IF GVL.g_stTrackingSimulation.Mode <> E_ApplicationSimulationMode.SIM_OFF AND GVL.g_stTrackingSimulation.VirtualEncoderEnable THEN 
	SMC_FreeEncoder.diEncoderPosition := diVirtualEncoderA; 
ELSE
	//SMC_FreeEncoder.diEncoderPosition := TO_DINT(AXIS_6.fActPosition);
	//SMC_FreeEncoder.diEncoderPosition :=AXIS_6.diActPosition;
// 	IF udiv < 400 THEN
// 		SMC_FreeEncoder.diEncoderPosition := SMC_FreeEncoder.diEncoderPosition - 10;
// 	END_IF
// 	IF udiv >= 400 THEN
// 		SMC_FreeEncoder.diEncoderPosition := SMC_FreeEncoder.diEncoderPosition - 11;
// 	END_IF
// 	IF udiv = 3 THEN
// 		SMC_FreeEncoder.diEncoderPosition := SMC_FreeEncoder.diEncoderPosition - 5;
// 	END_IF
// 	IF udiv = 4 THEN
// 		SMC_FreeEncoder.diEncoderPosition := SMC_FreeEncoder.diEncoderPosition - 5;
// 	END_IF
	IF GVL.Y[10] <> FALSE THEN
		SMC_FreeEncoder.diEncoderPosition := SMC_FreeEncoder.diEncoderPosition - GVL.g_HMI_PulsePerCycle_Set;
	END_IF;
END_IF;

IF udiv = 800 THEN udiv := 0; END_IF;
//=============================================================================
// 04. CONVEYOR RUNTIME STATUS
//-----------------------------------------------------------------------------
// Logical Axis SM_Drive_Logical đã được scale:
//     fActPosition = mm
//     fActVelocity = mm/s
//
// Mục đích:
//     - Cập nhật Status cho HMI.
//     - Làm nguồn dữ liệu chung cho Queue/Sensor/Vision.
//     - Tracking Manager đọc cùng một nguồn trạng thái Conveyor.
//=============================================================================

//-----------------------------------------------------------------------------
// 1. RAW POSITION / VELOCITY
//-----------------------------------------------------------------------------
GVL.g_aConveyorRuntime[1].Status.RawPosition :=
    LREAL_TO_REAL(SM_Drive_Logical.fActPosition);

GVL.g_aConveyorRuntime[1].Status.RawVelocity :=
    LREAL_TO_REAL(SM_Drive_Logical.fActVelocity);


//-----------------------------------------------------------------------------
// 2. POSITION THEO CHIỀU QUY ƯỚC CỦA APPLICATION
//-----------------------------------------------------------------------------
// DirectionSign:
//      +1 = giữ nguyên chiều Axis.
//      -1 = đảo chiều quy ước.
IF GVL.g_aConveyorRuntime[1].Config.DirectionSign >= 0 THEN
    GVL.g_aConveyorRuntime[1].Status.PositionMM :=
        LREAL_TO_REAL(SM_Drive_Logical.fActPosition);
ELSE
    GVL.g_aConveyorRuntime[1].Status.PositionMM :=
        -LREAL_TO_REAL(SM_Drive_Logical.fActPosition);
END_IF;


//-----------------------------------------------------------------------------
// 3. VELOCITY THEO CHIỀU QUY ƯỚC
//-----------------------------------------------------------------------------
IF GVL.g_aConveyorRuntime[1].Config.DirectionSign >= 0 THEN
    GVL.g_aConveyorRuntime[1].Status.VelocityMMs :=
        LREAL_TO_REAL(SM_Drive_Logical.fActVelocity);
ELSE
    GVL.g_aConveyorRuntime[1].Status.VelocityMMs :=
        -LREAL_TO_REAL(SM_Drive_Logical.fActVelocity);
END_IF;


//-----------------------------------------------------------------------------
// 4. GIỚI HẠN FILTER FACTOR 0.0 ... 1.0
//-----------------------------------------------------------------------------
IF GVL.g_aConveyorRuntime[1].Config.VelocityFilterFactor < 0.0 THEN
    GVL.g_aConveyorRuntime[1].Config.VelocityFilterFactor := 0.0;
ELSIF GVL.g_aConveyorRuntime[1].Config.VelocityFilterFactor > 1.0 THEN
    GVL.g_aConveyorRuntime[1].Config.VelocityFilterFactor := 1.0;
END_IF;


//-----------------------------------------------------------------------------
// 5. LOW-PASS FILTER VELOCITY
//-----------------------------------------------------------------------------
// FilterFactor = 1.0 : gần như lấy trực tiếp Velocity.
// FilterFactor nhỏ   : lọc mượt hơn nhưng phản ứng chậm hơn.
GVL.g_aConveyorRuntime[1].Status.FilteredVelocityMMs :=
    GVL.g_aConveyorRuntime[1].Status.FilteredVelocityMMs
    + GVL.g_aConveyorRuntime[1].Config.VelocityFilterFactor
    * (
        GVL.g_aConveyorRuntime[1].Status.VelocityMMs
        - GVL.g_aConveyorRuntime[1].Status.FilteredVelocityMMs
    );


//-----------------------------------------------------------------------------
// 6. ACCELERATION
//-----------------------------------------------------------------------------
// PRG_MultiToolTracking_A hiện chạy trong task 4 ms.
// a = Delta V / 0.004 s.
IF xConveyorRuntimeFirstScanA THEN

    GVL.g_aConveyorRuntime[1].Status.AccelerationMMs2 := 0.0;

    rConveyorVelocityPrevA :=
        GVL.g_aConveyorRuntime[1].Status.FilteredVelocityMMs;

    xConveyorRuntimeFirstScanA := FALSE;

ELSE

    GVL.g_aConveyorRuntime[1].Status.AccelerationMMs2 :=
        (
            GVL.g_aConveyorRuntime[1].Status.FilteredVelocityMMs
            - rConveyorVelocityPrevA
        ) / 0.004;

    rConveyorVelocityPrevA :=
        GVL.g_aConveyorRuntime[1].Status.FilteredVelocityMMs;

END_IF;


//-----------------------------------------------------------------------------
// 7. RUNNING / STANDSTILL / DIRECTION
//-----------------------------------------------------------------------------
IF ABS(GVL.g_aConveyorRuntime[1].Status.FilteredVelocityMMs)
    > GVL.g_aConveyorRuntime[1].Config.RunningThresholdMMs THEN

    GVL.g_aConveyorRuntime[1].Status.Running := TRUE;
    GVL.g_aConveyorRuntime[1].Status.Standstill := FALSE;

    IF GVL.g_aConveyorRuntime[1].Status.FilteredVelocityMMs > 0.0 THEN
        GVL.g_aConveyorRuntime[1].Status.Direction := 1;
    ELSE
        GVL.g_aConveyorRuntime[1].Status.Direction := -1;
    END_IF;

ELSE

    GVL.g_aConveyorRuntime[1].Status.Running := FALSE;
    GVL.g_aConveyorRuntime[1].Status.Standstill := TRUE;
    GVL.g_aConveyorRuntime[1].Status.Direction := 0;

END_IF;


//-----------------------------------------------------------------------------
// 8. VALID
//-----------------------------------------------------------------------------
GVL.g_aConveyorRuntime[1].Status.Valid :=
    GVL.g_aConveyorRuntime[1].Config.Enable;


//-----------------------------------------------------------------------------
// 9. ERROR LIMIT CHECK
//-----------------------------------------------------------------------------
GVL.g_aConveyorRuntime[1].Status.Error := FALSE;
GVL.g_aConveyorRuntime[1].Status.ErrorID := 0;

IF GVL.g_aConveyorRuntime[1].Config.MaxVelocityMMs > 0.0
AND ABS(GVL.g_aConveyorRuntime[1].Status.VelocityMMs)
    > GVL.g_aConveyorRuntime[1].Config.MaxVelocityMMs THEN

    GVL.g_aConveyorRuntime[1].Status.Error := TRUE;
    GVL.g_aConveyorRuntime[1].Status.ErrorID := 9001;

ELSIF GVL.g_aConveyorRuntime[1].Config.MaxAccelerationMMs2 > 0.0
AND ABS(GVL.g_aConveyorRuntime[1].Status.AccelerationMMs2)
    > GVL.g_aConveyorRuntime[1].Config.MaxAccelerationMMs2 THEN

    GVL.g_aConveyorRuntime[1].Status.Error := TRUE;
    GVL.g_aConveyorRuntime[1].Status.ErrorID := 9002;

END_IF;


rtCreateTestObjectA(CLK := GVL.g_xCreateTestTrackingObjectA);

IF rtCreateTestObjectA.Q THEN
    GVL.g_stTrackingQueue_A.NextObjectID := GVL.g_stTrackingQueue_A.NextObjectID + 1;
    IF GVL.g_stTrackingQueue_A.NextObjectID = 0 THEN GVL.g_stTrackingQueue_A.NextObjectID := 1; END_IF;

    GVL.g_stTrackingQueue_A.Objects[1].Valid := TRUE;
    GVL.g_stTrackingQueue_A.Objects[1].ObjectID := GVL.g_stTrackingQueue_A.NextObjectID;
    GVL.g_stTrackingQueue_A.Objects[1].ProductClassID := 1;
    GVL.g_stTrackingQueue_A.Objects[1].Reserved := FALSE;
    GVL.g_stTrackingQueue_A.Objects[1].ReservedToolID := 0;
    GVL.g_stTrackingQueue_A.Objects[1].CanPick := TRUE;
    GVL.g_stTrackingQueue_A.Objects[1].OrientationValid := TRUE;
    GVL.g_stTrackingQueue_A.Objects[1].VisionScore := 100.0;
    GVL.g_stTrackingQueue_A.Objects[1].State := E_TrackingObjectState.OBJ_READY;

    GVL.g_stTrackingQueue_A.Objects[1].VisionPos.X := 000.0;
    GVL.g_stTrackingQueue_A.Objects[1].VisionPos.Y := 0.0;
    GVL.g_stTrackingQueue_A.Objects[1].VisionPos.Z := 50.0;
    GVL.g_stTrackingQueue_A.Objects[1].VisionPos.A := 0.0;
	
	//-------------------------------------------------------------------------
	// OBJECT 1 - POSE CHUẨN TRONG HỆ CONVEYOR
	//-------------------------------------------------------------------------
	GVL.g_stTrackingQueue_A.Objects[1].PoseInConveyor.X := 000.0;
	GVL.g_stTrackingQueue_A.Objects[1].PoseInConveyor.Y := 0.0;
	GVL.g_stTrackingQueue_A.Objects[1].PoseInConveyor.Z := 50.0;
	GVL.g_stTrackingQueue_A.Objects[1].PoseInConveyor.A := 0.0;

	
	// Chốt vị trí Conveyor đúng thời điểm Object được tạo.
	GVL.g_stTrackingQueue_A.Objects[1].CaptureConveyorPositionMM :=
		REAL_TO_LREAL(GVL.g_aConveyorRuntime[1].Status.PositionMM);
	
	//---------------------------------------------------------------------
    // OBJECT 2
    //---------------------------------------------------------------------
    GVL.g_stTrackingQueue_A.NextObjectID :=
        GVL.g_stTrackingQueue_A.NextObjectID + 1;

    IF GVL.g_stTrackingQueue_A.NextObjectID = 0 THEN
        GVL.g_stTrackingQueue_A.NextObjectID := 1;
    END_IF;

    GVL.g_stTrackingQueue_A.Objects[2].Valid := TRUE;
    GVL.g_stTrackingQueue_A.Objects[2].ObjectID :=
        GVL.g_stTrackingQueue_A.NextObjectID;
    GVL.g_stTrackingQueue_A.Objects[2].ProductClassID := 1;
    GVL.g_stTrackingQueue_A.Objects[2].Reserved := FALSE;
    GVL.g_stTrackingQueue_A.Objects[2].ReservedToolID := 0;
    GVL.g_stTrackingQueue_A.Objects[2].CanPick := TRUE;
    GVL.g_stTrackingQueue_A.Objects[2].OrientationValid := TRUE;
    GVL.g_stTrackingQueue_A.Objects[2].VisionScore := 100.0;
    GVL.g_stTrackingQueue_A.Objects[2].State := E_TrackingObjectState.OBJ_READY;

    // Đặt cách Object 1 một khoảng để dễ quan sát.
    GVL.g_stTrackingQueue_A.Objects[2].VisionPos.X := 260.0;
    GVL.g_stTrackingQueue_A.Objects[2].VisionPos.Y := 0.0;
    GVL.g_stTrackingQueue_A.Objects[2].VisionPos.Z := 50.0;
    GVL.g_stTrackingQueue_A.Objects[2].VisionPos.A := 0.0;
	
	//-------------------------------------------------------------------------
	// OBJECT 2 - POSE CHUẨN TRONG HỆ CONVEYOR
	//-------------------------------------------------------------------------
	GVL.g_stTrackingQueue_A.Objects[2].PoseInConveyor.X := 260.0;
	GVL.g_stTrackingQueue_A.Objects[2].PoseInConveyor.Y := 0.0;
	GVL.g_stTrackingQueue_A.Objects[2].PoseInConveyor.Z := 50.0;
	GVL.g_stTrackingQueue_A.Objects[2].PoseInConveyor.A := 0.0;

	
	GVL.g_stTrackingQueue_A.Objects[2].CaptureConveyorPositionMM :=
		REAL_TO_LREAL(GVL.g_aConveyorRuntime[1].Status.PositionMM);

    GVL.g_stTrackingQueue_A.ValidCount := 2;
    GVL.g_stTrackingQueue_A.ActiveIndex := GVL.C_INVALID_INDEX;
	

//     GVL.g_stTrackingQueue_A.ValidCount := 1;
    GVL.g_stTrackingQueue_A.ActiveIndex := GVL.C_INVALID_INDEX;
END_IF;


//=============================================================================
// KHỞI TẠO CẤU HÌNH MẶC ĐỊNH CHO MULTI-TOOL ROBOT A
//-----------------------------------------------------------------------------
// Chỉ chạy một lần khi cấu hình chưa được khởi tạo hoặc khi người dùng yêu cầu
// khởi tạo lại. Không ghi đè cấu hình HMI trong mỗi vòng quét PLC.
//=============================================================================
IF (NOT GVL.g_xMultiToolConfigInitializedA OR GVL.g_xInitializeMultiToolConfigA) AND (1=2) THEN

    //-------------------------------------------------------------------------
    // TOOL 1
    //-------------------------------------------------------------------------
	GVL.g_aToolConfigA[1].Enable := TRUE;
	GVL.g_aToolConfigA[1].AllowTracking := TRUE;
	GVL.g_aToolConfigA[1].ToolID := 1;
	GVL.g_aToolConfigA[1].AllowedProductClassID := 0;
	

    //-------------------------------------------------------------------------
    // RECIPE 1 DÙNG CHO COMMISSIONING
    //-------------------------------------------------------------------------
    GVL.g_aMultiTrackRecipeA[1].Enable := TRUE;
    GVL.g_aMultiTrackRecipeA[1].RecipeID := 1;
    GVL.g_aMultiTrackRecipeA[1].ProductClassID := 0;
    GVL.g_aMultiTrackRecipeA[1].TargetPickCount := 1;
    GVL.g_aMultiTrackRecipeA[1].ToolEnableMask := DWORD#1;
	
	GVL.g_aToolConfigA[1].PickOffset.X := 0.0;
	GVL.g_aToolConfigA[1].PickOffset.Y := 0.0;
	GVL.g_aToolConfigA[1].PickOffset.Z := 50.0;
	GVL.g_aToolConfigA[1].PickOffset.A := 0.0;
	
	GVL.g_aToolConfigA[1].ApproachHeight := 20.0;
	GVL.g_aToolConfigA[1].UseUpDown := FALSE;
	GVL.g_aToolConfigA[1].UpDownStroke := 20.0;
	
	GVL.g_stTrackingConfig_A.RetractHeight := 20.0;
	
	
	//-------------------------------------------------------------------------
	// TOOL 2
	//-------------------------------------------------------------------------
	GVL.g_aToolConfigA[2].Enable := TRUE;
	GVL.g_aToolConfigA[2].AllowTracking := TRUE;
	GVL.g_aToolConfigA[2].ToolID := 2;
	GVL.g_aToolConfigA[2].AllowedProductClassID := 0;
	
	GVL.g_aToolConfigA[2].PickOffset.X := 0.0;
	GVL.g_aToolConfigA[2].PickOffset.Y := 0.0;
	GVL.g_aToolConfigA[2].PickOffset.Z := 50.0;
	GVL.g_aToolConfigA[2].PickOffset.A := 0.0;
	
	GVL.g_aToolConfigA[2].ApproachHeight := 20.0;
	
	// Có thể đặt khác Tool 1 để quan sát.
	GVL.g_aToolConfigA[2].UseUpDown := FALSE;
	GVL.g_aToolConfigA[2].UpDownStroke := 20.0;
	
	GVL.g_aToolConfigA[2].Priority := 2;


	//=============================================================================
	// DYNAMIC APPROACH
	//-----------------------------------------------------------------------------
	// Thông số thử nghiệm ban đầu. Có thể chỉnh lại trên HMI sau.
	//=============================================================================
	GVL.g_stTrackingConfig_A.Motion.Approach.Speed := 100.0;
	GVL.g_stTrackingConfig_A.Motion.Approach.Acceleration := 500.0;
	GVL.g_stTrackingConfig_A.Motion.Approach.Deceleration := 500.0;
	GVL.g_stTrackingConfig_A.Motion.Approach.Jerk := 1000.0;
	GVL.g_stTrackingConfig_A.Motion.Approach.BlendRadius := 0.0;
	
	GVL.g_stTrackingSimulation.VirtualEncoderStepPerCycle := -5;

    //-------------------------------------------------------------------------
    // ĐÁNH DẤU ĐÃ KHỞI TẠO
    //-------------------------------------------------------------------------
    GVL.g_xMultiToolConfigInitializedA := TRUE;
    GVL.g_xInitializeMultiToolConfigA := FALSE;

END_IF;

//=============================================================================
// PHỤC HỒI DỮ LIỆU COMMISSIONING KHI RESET MULTI-TOOL
//-----------------------------------------------------------------------------
// Chỉ dùng khi test Object cố định.
// Khi chạy Vision/Sensor thật, Object lỗi phải được loại bỏ hoặc nạp Object mới.
//=============================================================================
IF GVL.g_xMultiTrackResetTestA THEN


	//---------------------------------------------------------------------
    // RESET TOOL 1
    //---------------------------------------------------------------------
    GVL.g_aToolStatusA[1].Busy := FALSE;
    GVL.g_aToolStatusA[1].Occupied := FALSE;
    GVL.g_aToolStatusA[1].Error := FALSE;
    GVL.g_aToolStatusA[1].ErrorID := 0;
    GVL.g_aToolStatusA[1].HeldObjectID := 0;
    GVL.g_aToolStatusA[1].GripOK := FALSE;

    //---------------------------------------------------------------------
    // RESET TOOL 2
    //---------------------------------------------------------------------
    GVL.g_aToolStatusA[2].Busy := FALSE;
    GVL.g_aToolStatusA[2].Occupied := FALSE;
    GVL.g_aToolStatusA[2].Error := FALSE;
    GVL.g_aToolStatusA[2].ErrorID := 0;
    GVL.g_aToolStatusA[2].HeldObjectID := 0;
    GVL.g_aToolStatusA[2].GripOK := FALSE;
	
	// Comment lai vi dang test object thuc

//     //---------------------------------------------------------------------
//     // RESET OBJECT 1
//     //---------------------------------------------------------------------
//     GVL.g_stTrackingQueue_A.Objects[1].Valid := TRUE;
//     GVL.g_stTrackingQueue_A.Objects[1].CanPick := TRUE;
//     GVL.g_stTrackingQueue_A.Objects[1].Reserved := FALSE;
//     GVL.g_stTrackingQueue_A.Objects[1].ReservedToolID := 0;
//     GVL.g_stTrackingQueue_A.Objects[1].State :=
//         E_TrackingObjectState.OBJ_READY;
// 
//     //---------------------------------------------------------------------
//     // RESET OBJECT 2
//     //---------------------------------------------------------------------
//     GVL.g_stTrackingQueue_A.Objects[2].Valid := TRUE;
//     GVL.g_stTrackingQueue_A.Objects[2].CanPick := TRUE;
//     GVL.g_stTrackingQueue_A.Objects[2].Reserved := FALSE;
//     GVL.g_stTrackingQueue_A.Objects[2].ReservedToolID := 0;
//     GVL.g_stTrackingQueue_A.Objects[2].State :=
//         E_TrackingObjectState.OBJ_READY;
// 
//     GVL.g_stTrackingQueue_A.ValidCount := 2;
//     GVL.g_stTrackingQueue_A.ActiveIndex := GVL.C_INVALID_INDEX;

END_IF;

IF stCommandA.Reset THEN
    udiDebugCoreStartCountA := 0;
    udiDebugExecuteToCoreCountA := 0;
    udiDebugCoreRequestCountA := 0;

    xDebugCoreStartLatchedA := FALSE;
    xDebugExecuteToCoreLatchedA := FALSE;
    xDebugCoreRequestLatchedA := FALSE;
	GVL.g_xMultiTrackStartTestA := FALSE;
END_IF;

//=============================================================================
// 04. MULTI-TOOL CONTROLLER
//-----------------------------------------------------------------------------
// Controller đọc phản hồi của Core, SelectTool và ToolManager từ vòng quét trước.
//=============================================================================
fbControllerA(
    Command := stCommandA,
    CoreAccepted := fbCoreInterfaceA.Accepted,
    CoreBusy := fbCoreInterfaceA.Busy,
    CoreSyncOK := fbCoreInterfaceA.SyncOK,
    CorePCSInUse := fbCoreInterfaceA.PCSInUse,
    CoreReleased := fbCoreInterfaceA.Released,
    CoreError := fbCoreInterfaceA.Error,
    CoreErrorID := fbCoreInterfaceA.ErrorID,
    SelectToolDone := fbSelectToolA.Done,
    SelectToolError := fbSelectToolA.Error,
    SelectToolErrorID := fbSelectToolA.ErrorID,
    Queue := GVL.g_stTrackingQueue_A,
    ToolConfig := GVL.g_aToolConfigA,
    ToolStatus := GVL.g_aToolStatusA,
    Recipes := GVL.g_aMultiTrackRecipeA,
    Status := GVL.g_stMultiTrackStatusA
);


//=============================================================================
// MULTI-TOOL TRACKING RESULT LATCH
//=============================================================================

// Command mới được Controller nhận -> xóa kết quả command trước.
IF GVL.g_stMultiTrackStatusA.Accepted THEN
    GVL.g_xTrackOKA := FALSE;
    GVL.g_xTrackErrorA := FALSE;
    GVL.g_udiTrackErrorIDA := 0;
END_IF;


//-----------------------------------------------------------------------------
// TRACKING PICK HOÀN THÀNH ĐỦ SỐ LƯỢNG.
//-----------------------------------------------------------------------------
IF GVL.g_stMultiTrackStatusA.Done
AND NOT GVL.g_stMultiTrackStatusA.Error
AND GVL.g_stMultiTrackStatusA.PickedCount >= GVL.g_stMultiTrackStatusA.TargetPickCount THEN

    GVL.g_xTrackOKA := TRUE;
    GVL.g_xTrackErrorA := FALSE;
    GVL.g_udiTrackErrorIDA := 0;

    // Chốt CommandID của đúng lệnh vừa hoàn thành.
    GVL.g_udiTrackDoneCommandIDA :=
        GVL.g_stMultiTrackStatusA.ResponseCommandID;

END_IF;


//-----------------------------------------------------------------------------
// TRACKING ERROR.
//-----------------------------------------------------------------------------
IF GVL.g_stMultiTrackStatusA.Error THEN

    GVL.g_xTrackOKA := FALSE;
    GVL.g_xTrackErrorA := TRUE;
    GVL.g_udiTrackErrorIDA :=
        GVL.g_stMultiTrackStatusA.ErrorID;

END_IF;


//-----------------------------------------------------------------------------
// RESET.
//-----------------------------------------------------------------------------
IF stCommandA.Reset THEN

    GVL.g_xTrackOKA := FALSE;
    GVL.g_xTrackErrorA := FALSE;
    GVL.g_udiTrackErrorIDA := 0;
    GVL.g_udiTrackDoneCommandIDA := 0;

END_IF;



//=============================================================================
// 05. TRACKING CORE INTERFACE
//-----------------------------------------------------------------------------
// Interface giữ Execute cho Tracking Core và chỉ hạ sau khi PCS đã release.
//=============================================================================
fbCoreInterfaceA(
    Enable := TRUE,
    Reset := fbControllerA.CoreReset,
    Abort := fbControllerA.CoreAbort,
    StartTracking := fbControllerA.CoreStart,
    ReleaseTracking := fbControllerA.CoreRelease,
    ObjectIndex := fbControllerA.CoreObjectIndex,
    ToolID := fbControllerA.CoreToolID,
    PickOffset := fbControllerA.CorePickOffset,
    ApproachHeight := fbControllerA.CoreApproachHeight,
	PickSurfaceHeightMM := fbControllerA.CorePickSurfaceHeightMM,
    CoreAccepted := GVL.g_stTrackingRuntime_A.Response.Accepted,
	CoreBusy := GVL.g_stTrackingRuntime_A.Response.Busy,
	CoreSyncOK := fbTrackingManagerA.SyncOK,
	CorePCSInUse := GVL.g_stTrackingRuntime_A.PCSInfo.InUse,
	CoreReleased := fbTrackingManagerA.Released,
	CoreError := GVL.g_stTrackingRuntime_A.Response.Error,
	CoreErrorID := GVL.g_stTrackingRuntime_A.Response.ErrorID,
	UseUpDown := fbControllerA.CoreUseUpDown,
	UpDownStroke := fbControllerA.CoreUpDownStroke,
);


//=============================================================================
// 06. CHỌN TOOL/TCP ROBOT A
//-----------------------------------------------------------------------------
// FB_SelectRobotTool phải gọi SMC_GroupSetTool thực tế, không dùng placeholder.
//=============================================================================
fbSelectToolA(
    Execute := fbControllerA.SelectToolExecute,
    Reset := stCommandA.Reset,
    ToolID := fbControllerA.SelectToolID
);


// xTrackingRequestValid :=
//     fbCoreInterfaceA.ExecuteToCore
//     AND fbCoreInterfaceA.ActiveObjectIndex >= 1
//     AND fbCoreInterfaceA.ActiveObjectIndex <= GVL.C_MAX_TRACK_OBJECTS
//     AND GVL.g_stTrackingQueue_A.Objects[fbCoreInterfaceA.ActiveObjectIndex].Valid;
	
xCoreRequestValid := fbCoreInterfaceA.ExecuteToCore
AND fbCoreInterfaceA.ActiveObjectIndex >= 1
AND fbCoreInterfaceA.ActiveObjectIndex <= GVL.C_MAX_TRACK_OBJECTS
AND GVL.g_stTrackingQueue_A.Objects[fbCoreInterfaceA.ActiveObjectIndex].Valid;

rtDebugCoreStartA(CLK := fbControllerA.CoreStart);
rtDebugExecuteToCoreA(CLK := fbCoreInterfaceA.ExecuteToCore);
rtDebugCoreRequestValidA(CLK := xCoreRequestValid);

IF rtDebugCoreStartA.Q THEN
    udiDebugCoreStartCountA := udiDebugCoreStartCountA + 1;
    xDebugCoreStartLatchedA := TRUE;
END_IF;

IF rtDebugExecuteToCoreA.Q THEN
    udiDebugExecuteToCoreCountA := udiDebugExecuteToCoreCountA + 1;
    xDebugExecuteToCoreLatchedA := TRUE;
END_IF;

IF rtDebugCoreRequestValidA.Q THEN
    udiDebugCoreRequestCountA := udiDebugCoreRequestCountA + 1;
    xDebugCoreRequestLatchedA := TRUE;
END_IF;


//=============================================================================
// 07. TRACKING CORE
//-----------------------------------------------------------------------------
// Multi-tool mode luôn dùng UseExternalSelection = TRUE.
// Controller đã chọn ObjectIndex và PickOffset theo Tool.
//=============================================================================
fbTrackingManagerA(
    Execute := xCoreRequestValid,
    Reset := fbCoreInterfaceA.ResetToCore OR stCommandA.Reset,
    Config := GVL.g_stTrackingConfig_A,
    ConveyorConfig := GVL.g_aConveyorRuntime[1].Config,
    ConveyorStatus := GVL.g_aConveyorRuntime[1].Status,
    ConveyorOrigin := stConveyorOriginA,
    VacuumOK := FALSE,
    MotionAccepted := GVL.g_xTrackingMotionAccepted,
    MotionBusy := GVL.g_xTrackingMotionBusy,
    MotionDone := GVL.g_xTrackingMotionDone,
    MotionError := GVL.g_xTrackingMotionError,
    MotionErrorID := GVL.g_udiTrackingMotionErrorID,
    MotionAbortDone := GVL.g_xTrackingMotionAbortDone,
    TestFixedObjectMode := FALSE,
    FixedObjectPosition := stFixedObjectPositionA,
    UseExternalSelection := TRUE,
    ExternalObjectIndex := fbCoreInterfaceA.ActiveObjectIndex,
    ExternalPickOffset := fbCoreInterfaceA.ActivePickOffset,
    ExternalApproachHeight := fbCoreInterfaceA.ActiveApproachHeight,
    PickerSafe := fbCoreInterfaceA.PickerSafeToCore,
    Queue := GVL.g_stTrackingQueue_A,
    Runtime := GVL.g_stTrackingRuntime_A,
	ExternalUseUpDown := fbCoreInterfaceA.ActiveUseUpDown,
	ExternalUpDownStroke := fbCoreInterfaceA.ActiveUpDownStroke,
	ExternalPickSurfaceHeightMM := fbCoreInterfaceA.ActivePickSurfaceHeightMM,
);


//=============================================================================
// 08. MAP PHẢN HỒI TRACKING CORE
//-----------------------------------------------------------------------------
// Các biến này được FB_TrackingCoreInterface_A đọc ở vòng quét tiếp theo.
//=============================================================================
GVL.g_xTrackingCoreAcceptedA := GVL.g_stTrackingRuntime_A.Response.Accepted;
GVL.g_xTrackingCoreBusyA := GVL.g_stTrackingRuntime_A.Response.Busy;
GVL.g_xTrackingCoreSyncOKA := fbTrackingManagerA.SyncOK;
GVL.g_xTrackingCorePCSInUseA := GVL.g_stTrackingRuntime_A.PCSInfo.InUse;
GVL.g_xTrackingCoreReleasedA := fbTrackingManagerA.Released;
GVL.g_xTrackingCoreErrorA := GVL.g_stTrackingRuntime_A.Response.Error;
GVL.g_udiTrackingCoreErrorIDA := GVL.g_stTrackingRuntime_A.Response.ErrorID;


//=============================================================================
// 09. MOTION QUEUE ADAPTER
//-----------------------------------------------------------------------------
// Chỉ instance này được đưa motion Tracking vào Motion Queue Robot A.
//=============================================================================
fbMotionAdapterA(
    Enable := TRUE,
    Reset := fbCoreInterfaceA.ResetToCore OR stCommandA.Reset,
    Request := fbTrackingManagerA.MotionRequest,
    Abort := fbTrackingManagerA.MotionAbort,
    Target := fbTrackingManagerA.MotionTarget,
    Speed := fbTrackingManagerA.MotionSpeed,
    Acceleration := fbTrackingManagerA.MotionAcceleration,
    Deceleration := fbTrackingManagerA.MotionDeceleration,
    Jerk := fbTrackingManagerA.MotionJerk,
    BlendRadius := fbTrackingManagerA.MotionBlendRadius,
    CoordSystem := fbTrackingManagerA.MotionCoordSystem,
    Command := fbTrackingManagerA.MotionCommand,
    LogicSimulation := GVL.g_stTrackingSimulation.Mode = E_ApplicationSimulationMode.SIM_LOGIC_ONLY,
    LogicMotionDuration := GVL.g_stTrackingSimulation.LogicMotionDuration,
    Accepted => GVL.g_xTrackingMotionAccepted,
    Busy => GVL.g_xTrackingMotionBusy,
    Done => GVL.g_xTrackingMotionDone,
    Error => GVL.g_xTrackingMotionError,
    ErrorID => GVL.g_udiTrackingMotionErrorID,
    AbortDone => GVL.g_xTrackingMotionAbortDone
);


//=============================================================================
// 10. PHÂN PHỐI COMMAND TỚI TỪNG TOOL MANAGER
//-----------------------------------------------------------------------------
// Chỉ Tool có ToolID trùng Command mới nhận Execute.
// Các Tool còn lại vẫn được gọi mỗi vòng quét để duy trì Runtime và Output.
//=============================================================================
FOR uiTool := 1 TO GVL.C_MAX_TOOLS DO
	
	// Tất cả OUTPUT mặc định Active HIGH.
	GVL.g_aToolConfigA[uiTool].IO.DownDOActiveLevel := TRUE;
	GVL.g_aToolConfigA[uiTool].IO.UpDOActiveLevel := TRUE;
	GVL.g_aToolConfigA[uiTool].IO.GripDOActiveLevel := TRUE;
	GVL.g_aToolConfigA[uiTool].IO.ReleaseDOActiveLevel := TRUE;
	
	// Tất cả INPUT feedback mặc định Active HIGH.
	GVL.g_aToolConfigA[uiTool].IO.DownOKDIActiveLevel := TRUE;
	GVL.g_aToolConfigA[uiTool].IO.UpOKDIActiveLevel := TRUE;
	GVL.g_aToolConfigA[uiTool].IO.GripOKDIActiveLevel := TRUE;
	GVL.g_aToolConfigA[uiTool].IO.PartPresentDIActiveLevel := TRUE;
	
    astToolCommandA[uiTool].Execute := FALSE;
    astToolCommandA[uiTool].Reset := stCommandA.Reset;
    astToolCommandA[uiTool].Abort := stCommandA.Abort;
    astToolCommandA[uiTool].CommandID := 0;
    astToolCommandA[uiTool].ToolID := GVL.g_aToolConfigA[uiTool].ToolID;
    astToolCommandA[uiTool].CommandType := E_ToolCommandType.NONE;
    astToolCommandA[uiTool].ObjectID := 0;

    //IF fbControllerA.ToolCommand.ToolID = GVL.g_aToolConfigA[uiTool].ToolID THEN astToolCommandA[uiTool] := fbControllerA.ToolCommand; END_IF;
	
//-------------------------------------------------------------------------
	// ƯU TIÊN 1: Command từ MultiTool Tracking Controller.
	//-------------------------------------------------------------------------
	IF fbControllerA.ToolCommand.Execute
	AND fbControllerA.ToolCommand.ToolID = GVL.g_aToolConfigA[uiTool].ToolID THEN
	
		astToolCommandA[uiTool] := fbControllerA.ToolCommand;
	
	
	//-------------------------------------------------------------------------
	// ƯU TIÊN 2: Command Tool độc lập từ Interpreter.
	// Chỉ chạy khi Controller không phát Tool Command.
	//-------------------------------------------------------------------------
	ELSIF GVL.g_stInterpreterToolCommandA.Execute
	AND GVL.g_stInterpreterToolCommandA.ToolID = GVL.g_aToolConfigA[uiTool].ToolID THEN
	
		astToolCommandA[uiTool] :=
			GVL.g_stInterpreterToolCommandA;
	
	END_IF;

    fbToolManagerA[uiTool](
        Enable := GVL.g_aToolConfigA[uiTool].Enable,
        Command := astToolCommandA[uiTool],
        Config := GVL.g_aToolConfigA[uiTool],
        Status := GVL.g_aToolStatusA[uiTool]
    );
END_FOR;


//=============================================================================
// 11. BIẾN GIÁM SÁT HMI / DEBUG
//=============================================================================
GVL.g_xMultiTrackCoreExecuteA := fbCoreInterfaceA.ExecuteToCore;
GVL.g_xMultiTrackCoreResetA := fbCoreInterfaceA.ResetToCore;
GVL.g_xMultiTrackCoreAbortA := fbCoreInterfaceA.AbortToCore;
GVL.g_xMultiTrackPickerSafeA := fbCoreInterfaceA.PickerSafeToCore;
GVL.g_uiMultiTrackObjectIndexA := fbCoreInterfaceA.ActiveObjectIndex;
GVL.g_uiMultiTrackToolIDA := fbCoreInterfaceA.ActiveToolID;
GVL.g_stMultiTrackPickOffsetA := fbCoreInterfaceA.ActivePickOffset;
GVL.g_rMultiTrackApproachHeightA := fbCoreInterfaceA.ActiveApproachHeight;
GVL.g_xSelectToolExecuteA := fbControllerA.SelectToolExecute;
GVL.g_uiSelectToolIDA := fbControllerA.SelectToolID;
GVL.g_stSelectToolTCPA := fbControllerA.SelectToolTCP;
GVL.g_xSelectToolDoneA := fbSelectToolA.Done;
GVL.g_xSelectToolErrorA := fbSelectToolA.Error;
GVL.g_udiSelectToolErrorIDA := fbSelectToolA.ErrorID;


//=============================================================================
// 12. OUTPUT CŨ CỦA TRACKING CORE
//-----------------------------------------------------------------------------
// Multi-tool mode không dùng VacuumCommand/BlowCommand; giữ map để debug.
//=============================================================================
GVL.g_xTrackingVacuumOutput := fbTrackingManagerA.VacuumCommand;
GVL.g_xTrackingBlowOutput := fbTrackingManagerA.BlowCommand;

END_PROGRAM

// Just_Motion_Control_x86_64_Linux_SM_WV/Application/FB_/TOOL/FB_SelectRobotTool
FUNCTION_BLOCK FB_SelectRobotTool
VAR_INPUT

    // Xung Execute.
    Execute : BOOL;

    // Reset FB.
    Reset : BOOL;

    // ToolID cần chọn.
    ToolID : UINT;

    

END_VAR

VAR_OUTPUT

    // Tool đã được chọn.
    Done : BOOL;

    // FB đang xử lý.
    Busy : BOOL;

    // FB lỗi.
    Error : BOOL;

    // Mã lỗi.
    ErrorID : UDINT;

END_VAR

VAR

    // Bắt cạnh Execute.
    rtExecute : R_TRIG;

    // TODO:
    // Khai báo instance SMC_GroupSetTool đúng theo version thư viện.
    fbGroupSetTool : SMC_GroupSetTool;
	xExecuteTool : BOOL;
	// RequestID thuộc transaction hiện tại.
	udiMyRequestID : UDINT := 0;

END_VAR

//=============================================================================
// FB_SelectRobotTool
//-----------------------------------------------------------------------------
// ToolID = Number_Tool.
// Không gọi SMC_GroupSetTool tại đây.
// POU_COORDINATE_ là nơi duy nhất Apply TCP vào SCARA_A.
//=============================================================================

Done := FALSE;


//=============================================================================
// RESET
//=============================================================================
IF Reset THEN
    Busy := FALSE;
    Error := FALSE;
    ErrorID := 0;
    udiMyRequestID := 0;
    RETURN;
END_IF;


//=============================================================================
// DETECT EXECUTE
//=============================================================================
rtExecute(CLK := Execute);


//=============================================================================
// TẠO YÊU CẦU CHỌN / APPLY TOOL
//=============================================================================
IF rtExecute.Q AND NOT Busy THEN

    Busy := TRUE;
    Error := FALSE;
    ErrorID := 0;

    //---------------------------------------------------------------------
    // ToolID chính là Number_Tool.
    //
    // ToolID = 0 : No Tool Offset.
    // ToolID = 1 : Tool 1.
    // ToolID = 2 : Tool 2...
    //---------------------------------------------------------------------
    GVL.RB_A.Number_Tool := ToolID;

    //---------------------------------------------------------------------
    // Luôn tạo Request mới.
    // Nhờ vậy cùng ToolID nhưng TCP đã thay đổi vẫn được Apply lại.
    //---------------------------------------------------------------------
    GVL.g_udiRobotAToolApplyRequestA := GVL.g_udiRobotAToolApplyRequestA + 1;
    IF GVL.g_udiRobotAToolApplyRequestA = 0 THEN GVL.g_udiRobotAToolApplyRequestA := 1; END_IF;

    // Chốt Request của transaction này.
    udiMyRequestID := GVL.g_udiRobotAToolApplyRequestA;

END_IF;


//=============================================================================
// CHỜ KẾT QUẢ TỪ POU_COORDINATE_
//=============================================================================
IF Busy THEN

    //---------------------------------------------------------------------
    // APPLY ERROR
    //---------------------------------------------------------------------
    IF GVL.g_xRobotAToolApplyError THEN
        Busy := FALSE;
        Error := TRUE;
        ErrorID := GVL.g_udiRobotAToolApplyErrorID;

    //---------------------------------------------------------------------
    // APPLY DONE
    //---------------------------------------------------------------------
    ELSIF udiMyRequestID <> 0
    AND GVL.g_udiRobotAToolAppliedRequestA = udiMyRequestID THEN
        Busy := FALSE;
        Error := FALSE;
        ErrorID := 0;
        Done := TRUE;
    END_IF;

END_IF;





// (*
// ===============================================================================
// FUNCTION BLOCK
//     FB_SelectRobotTool
// 
// DESCRIPTION
//     Wrapper chọn Tool/TCP cho Robot.
// 
// TODO INTEGRATIONđ
//     Thay phần Logic-Only Placeholder bằng SMC_GroupSetTool đang có
//     trong project hiện tại.
// 
// EXPECTED FLOW
//     Execute rising edge
//         -> Call SMC_GroupSetTool
//         -> Wait Done/Error
//         -> Return Done/Error
// ===============================================================================
// *)
// 
// //=============================================================================
// // DEFAULT PULSE OUTPUT
// //=============================================================================
// Done := FALSE;
// 
// 
// //=============================================================================
// // RESET
// //=============================================================================
// IF Reset THEN
// 
//     Busy := FALSE;
// 
//     Error := FALSE;
//     ErrorID := 0;
// 
//     RETURN;
// 
// END_IF;
// 
// 
// //=============================================================================
// // DETECT EXECUTE
// //=============================================================================
// rtExecute(CLK := Execute);
// 
// 
// //=============================================================================
// // START TOOL SELECTION
// //=============================================================================
// IF rtExecute.Q AND NOT Busy THEN
// 
//     Busy := TRUE;
// 
//     Error := FALSE;
//     ErrorID := 0;
// 
// 
//     //=========================================================================
//     // TODO: CALL SMC_GROUPSETTOOL HERE
//     //-------------------------------------------------------------------------
//     // Ví dụ logic:
//     //
// 	fbGroupSetTool(
// 		Execute   := TRUE,
// 		AxisGroup := SCARA_A,
// 		ToolOffset := F_ConvertToolTCP(ToolTCP)
// 	);
// 	
// 	IF fbGroupSetTool.Done THEN
// 		Busy := FALSE;
// 		Done := TRUE;
// 	END_IF;
// 	
// 	IF fbGroupSetTool.Error THEN
// 		Busy := FALSE;
// 		Error := TRUE;
// 		ErrorID := fbGroupSetTool.ErrorID;
// 	END_IF;
//     //=========================================================================
// 
// 
// //     //-------------------------------------------------------------------------
// //     // LOGIC-ONLY PLACEHOLDER
// //     //-------------------------------------------------------------------------
// //     // Xóa hai dòng dưới sau khi nối SMC_GroupSetTool thực tế.
// //     Busy := FALSE;
// //     Done := TRUE;
// 
// END_IF;
//

END_FUNCTION_BLOCK

// Just_Motion_Control_x86_64_Linux_SM_WV/Application/FC_/Tool/F_ConvertToolTCP
FUNCTION F_ConvertToolTCP : SM3_Robotics.MC_COORD_REF
VAR_INPUT
	TOOLTCP      : ST_POS;
END_VAR

F_ConvertToolTCP.X := TO_LREAL(TOOLTCP.X);
F_ConvertToolTCP.Y := TO_LREAL(TOOLTCP.Y);
F_ConvertToolTCP.Z := TO_LREAL(TOOLTCP.Z);
F_ConvertToolTCP.A := TO_LREAL(TOOLTCP.A);
F_ConvertToolTCP.B := TO_LREAL(0);
F_ConvertToolTCP.C := TO_LREAL(0);

END_FUNCTION

// Just_Motion_Control_x86_64_Linux_SM_WV/Application/FB_/ConveyorTrack/FB_TrackingCoreInterface_A
FUNCTION_BLOCK FB_TrackingCoreInterface_A
VAR_INPUT
    Enable : BOOL;
    Reset : BOOL;
    Abort : BOOL;
    StartTracking : BOOL;
    ReleaseTracking : BOOL;
    ObjectIndex : UINT;
    ToolID : UINT;
    PickOffset : ST_POS;
    ApproachHeight : REAL;
	PickSurfaceHeightMM : REAL;
    CoreAccepted : BOOL;
    CoreBusy : BOOL;
    CoreSyncOK : BOOL;
    CorePCSInUse : BOOL;
    CoreReleased : BOOL;
    CoreError : BOOL;
    CoreErrorID : UDINT;
	UseUpDown : BOOL;
	UpDownStroke : REAL;
END_VAR
VAR_OUTPUT
    ExecuteToCore : BOOL;
    ResetToCore : BOOL;
    AbortToCore : BOOL;
    PickerSafeToCore : BOOL;
    ActiveObjectIndex : UINT;
    ActiveToolID : UINT;
    ActivePickOffset : ST_POS;
    ActiveApproachHeight : REAL;
	ActivePickSurfaceHeightMM : REAL;
    Accepted : BOOL;
    Busy : BOOL;
    SyncOK : BOOL;
    PCSInUse : BOOL;
    Released : BOOL;
    Error : BOOL;
    ErrorID : UDINT;
	ActiveUseUpDown : BOOL;
	ActiveUpDownStroke : REAL;
END_VAR
VAR
    rtStart : R_TRIG;
    xRequestLatched : BOOL := FALSE;
	// TRUE sau khi Controller yêu cầu kết thúc Tracking.
	xReleaseRequested : BOOL := FALSE;
	
	// Bắt cạnh lên của tín hiệu CoreReleased.
	rtCoreReleased : R_TRIG;
	xCoreWasBusy : BOOL := FALSE;
	xCoreWasInUse : BOOL := FALSE;	
	
	
END_VAR

(*
===============================================================================
FB_TrackingCoreInterface_A

MỤC ĐÍCH
    Chuẩn hóa handshake giữa MultiTool Controller và
    FB_CONVEYOR_TRACKING_MANAGER.
===============================================================================
*)

//=============================================================================
// BẮT CẠNH TÍN HIỆU
//=============================================================================
rtStart(CLK := StartTracking);
rtCoreReleased(CLK := CoreReleased);


//=============================================================================
// OUTPUT MẶC ĐỊNH MỖI VÒNG QUÉT
//=============================================================================
ResetToCore := FALSE;
AbortToCore := FALSE;
Released := FALSE;

Accepted := CoreAccepted AND xRequestLatched;
Busy := CoreBusy AND xRequestLatched;
SyncOK := CoreSyncOK AND xRequestLatched;
PCSInUse := CorePCSInUse AND xRequestLatched;
Error := CoreError AND xRequestLatched;


IF Error THEN
    ErrorID := CoreErrorID;
ELSE
    ErrorID := 0;
END_IF;


//=============================================================================
// RESET / DISABLE
//=============================================================================
IF Reset OR NOT Enable THEN
    ExecuteToCore := FALSE;
    ResetToCore := Reset;
    AbortToCore := FALSE;
    PickerSafeToCore := FALSE;
    Released := FALSE;

    xRequestLatched := FALSE;
    xReleaseRequested := FALSE;
    xCoreWasBusy := FALSE;
    xCoreWasInUse := FALSE;

    ActiveObjectIndex := 0;
    ActiveToolID := 0;
    ActivePickOffset.X := 0.0;
    ActivePickOffset.Y := 0.0;
    ActivePickOffset.Z := 0.0;
    ActivePickOffset.A := 0.0;
    ActiveApproachHeight := 0.0;

    Accepted := FALSE;
    Busy := FALSE;
    SyncOK := FALSE;
    PCSInUse := FALSE;
    Error := FALSE;
    ErrorID := 0;
	ActiveUseUpDown := FALSE;
	ActiveUpDownStroke := 0.0;
	ActivePickSurfaceHeightMM := 0.0;

    RETURN;
END_IF;


//=============================================================================
// ABORT
//=============================================================================
IF Abort THEN
    ExecuteToCore := FALSE;
    ResetToCore := FALSE;
    AbortToCore := TRUE;
    PickerSafeToCore := FALSE;
    Released := FALSE;

    xRequestLatched := FALSE;
    xReleaseRequested := FALSE;
    xCoreWasBusy := FALSE;
    xCoreWasInUse := FALSE;

    Accepted := FALSE;
    Busy := FALSE;
    SyncOK := FALSE;
    PCSInUse := FALSE;
	
	ActiveUseUpDown := FALSE;
	ActiveUpDownStroke := 0.0;
    RETURN;
END_IF;


//=============================================================================
// START TRACKING REQUEST
//=============================================================================
IF rtStart.Q AND NOT xRequestLatched THEN
    IF ObjectIndex >= 1
    AND ObjectIndex <= GVL.C_MAX_TRACK_OBJECTS THEN

        ActiveObjectIndex := ObjectIndex;
        ActiveToolID := ToolID;
        ActivePickOffset := PickOffset;
        ActiveApproachHeight := ApproachHeight;
		ActivePickSurfaceHeightMM := PickSurfaceHeightMM;
        ActiveUseUpDown := UseUpDown;
        ActiveUpDownStroke := UpDownStroke;

        xRequestLatched := TRUE;
        xReleaseRequested := FALSE;
    END_IF;

END_IF;


//=============================================================================
// GIỮ EXECUTE TRONG TOÀN BỘ REQUEST
//=============================================================================
ExecuteToCore := xRequestLatched;

// Nhận yêu cầu release từ Controller.
IF ReleaseTracking AND xRequestLatched THEN
    xReleaseRequested := TRUE;
END_IF;

PickerSafeToCore := xRequestLatched AND xReleaseRequested;

// Chỉ đóng request khi Manager đã phát Released.
IF rtCoreReleased.Q
AND xRequestLatched
AND xReleaseRequested THEN
    Released := TRUE;
    ExecuteToCore := FALSE;
    PickerSafeToCore := FALSE;

    xRequestLatched := FALSE;
    xReleaseRequested := FALSE;

    ActiveObjectIndex := 0;
    ActiveToolID := 0;
	
	ActiveUseUpDown := FALSE;
	ActiveUpDownStroke := 0.0;
	
END_IF;

END_FUNCTION_BLOCK

// Just_Motion_Control_x86_64_Linux_SM_WV/Application/FB_/ConveyorTrack/FB_CONVEYOR_TRACKING_MANAGER
FUNCTION_BLOCK FB_CONVEYOR_TRACKING_MANAGER
VAR_INPUT
    Execute : BOOL;
    Reset : BOOL;
    Config : ST_TRACKING_CONFIG;
    ConveyorConfig : ST_CONVEYOR_CONFIG;
    ConveyorStatus : ST_CONVEYOR_STATUS;
    ConveyorOrigin : MC_COORD_REF;
    VacuumOK : BOOL;
    MotionAccepted : BOOL;
    MotionBusy : BOOL;
    MotionDone : BOOL;
    MotionError : BOOL;
    MotionErrorID : UDINT;
    MotionAbortDone : BOOL;
    TestFixedObjectMode : BOOL;
    FixedObjectPosition : MC_COORD_REF;

    // Multi-tool external control.
    UseExternalSelection : BOOL;
    ExternalObjectIndex : UINT;
    ExternalPickOffset : ST_POS;
    ExternalApproachHeight : REAL;
    PickerSafe : BOOL;
	ExternalUseUpDown : BOOL;
	ExternalUpDownStroke : REAL;
	// Chiều cao mặt cần hút của sản phẩm.
	// Được lấy từ Recipe khi chạy MultiTool.
	ExternalPickSurfaceHeightMM : REAL;
END_VAR

VAR_OUTPUT
    VacuumCommand : BOOL;
    BlowCommand : BOOL;
    TrackingActive : BOOL;
    MotionRequest : BOOL;
    MotionAbort : BOOL;
    MotionTarget : ST_POS;
    MotionSpeed : REAL;
    MotionAcceleration : REAL;
    MotionDeceleration : REAL;
    MotionJerk : REAL;
    MotionBlendRadius : REAL;
    MotionCoordSystem : E_AppCoordSystem;
    MotionCommand : UINT;

    // Multi-tool handshake.
    SyncOK : BOOL;
    Released : BOOL;
END_VAR

VAR_IN_OUT
    Queue : ST_TRACKING_QUEUE;
    Runtime : ST_TRACKING_RUNTIME;
END_VAR

VAR
    fbTrackBelt : MC_TrackConveyorBelt;
    xTrackExecute : BOOL;
    uiSelectedIndex : UINT;
    stSelectedObject : ST_TRACKING_OBJECT;
    xMotionIssued : BOOL;
    xMotionRequestPending : BOOL;
    xMotionActive : BOOL;
    xVacuumCaptured : BOOL;
    tonPickDelay : TON;
    tonVacuumTimeout : TON;
    tonBlow : TON;
    stConveyorOriginSMC : MC_COORD_REF;
    stInitialObjectSMC : MC_COORD_REF;
    stExitPCSTarget : ST_POS;
    xExitPCSTargetValid : BOOL := FALSE;
    rExitPCSOffsetZ : REAL := 5.0;
	rExitPCSOffsetX : REAL := 15.0;
    rExitPCSMaxZ : REAL := 320.0;
	stToolSyncPos : ST_POS;
	xPickPositionReady : BOOL;
	xPickerSafeArmed : BOOL;
	xMotionDoneArmed : BOOL;
	xPickMotionBusySeen : BOOL; //xác nhận lệnh xuống Pick thực sự chạy.
	xRetractMotionBusySeen : BOOL; // xác nhận lệnh nâng Retract thực sự chạy.
	lrConveyorDeltaAtPCS : LREAL;
END_VAR
VAR
    // TRUE khi đã chụp vị trí Conveyor cho lần tạo PCS hiện tại.
    xPCSStartCaptured : BOOL;

    // Vị trí Conveyor tại thời điểm chuẩn bị phát cạnh Track Execute.
    lrConveyorPosAtPCSStart : LREAL;

    // Conveyor đã dịch từ lúc Object được Sensor/Vision Capture tới lúc tạo PCS.
    lrDeltaCaptureToPCS : LREAL;
END_VAR

(*
===============================================================================
FB_CONVEYOR_TRACKING_MANAGER - MULTI-TOOL CORE V2
===============================================================================
- Giữ chế độ Tracking Pick cũ khi UseExternalSelection = FALSE.
- Thêm chế độ Multi-tool khi UseExternalSelection = TRUE.
- Multi-tool Core chỉ tạo PCS, chạy Approach, chờ PickerSafe và thoát PCS.
- Tool DOWN/GRIP/UP do FB_ToolManager bên ngoài điều khiển.
===============================================================================
*)

//=============================================================================
// 01. CHUYỂN ĐỔI GỐC CONVEYOR SANG KIỂU POSE CỦA SOFTMOTION
//=============================================================================

// Chuyển tọa độ X của gốc conveyor.
stConveyorOriginSMC.X := ConveyorOrigin.X;
// Chuyển tọa độ Y của gốc conveyor.
stConveyorOriginSMC.Y := ConveyorOrigin.Y;
// Chuyển tọa độ Z của gốc conveyor.
stConveyorOriginSMC.Z := ConveyorOrigin.Z;
// Chuyển góc A của gốc conveyor.
stConveyorOriginSMC.A := ConveyorOrigin.A;
// Chuyển góc B của gốc conveyor.
stConveyorOriginSMC.B := 0.0;
// Chuyển góc C của gốc conveyor.
stConveyorOriginSMC.C := 0.0;

//=============================================================================
// 02. CHUYỂN ĐỔI POSE OBJECT BAN ĐẦU SANG KIỂU SOFTMOTION
//=============================================================================

// Chuyển tọa độ X của object ban đầu.
stInitialObjectSMC.X := Runtime.PCSInfo.InitialObjectPos.X;

// Chuyển tọa độ Y của object ban đầu.
stInitialObjectSMC.Y := Runtime.PCSInfo.InitialObjectPos.Y;

// Chuyển tọa độ Z của object ban đầu.
stInitialObjectSMC.Z := Runtime.PCSInfo.InitialObjectPos.Z;

// Chuyển góc A của object ban đầu.
stInitialObjectSMC.A := Runtime.PCSInfo.InitialObjectPos.A;

// // Chuyển góc B của object ban đầu.
// stInitialObjectSMC.B :=
//     REAL_TO_LREAL(Runtime.PCSInfo.InitialObjectPos.B);
// 
// // Chuyển góc C của object ban đầu.
// stInitialObjectSMC.C :=
//     REAL_TO_LREAL(Runtime.PCSInfo.InitialObjectPos.C);

//=============================================================================
// 03. GỌI MC_TrackConveyorBelt MỖI VÒNG QUÉT
//-----------------------------------------------------------------------------
// Không đặt lời gọi này chỉ trong một CASE state.
// Không hạ xTrackExecute ngay khi fbTrackBelt.Done.
//=============================================================================

fbTrackBelt(
    // Axis Group robot SCARA hiện tại.
    AxisGroup := SCARA_A,

    // Logical Axis conveyor đã chạy trong chương trình test.
    ConveyorBelt := SM_Drive_Logical,

    // Execute nội bộ điều khiển vòng đời PCS.
    Execute := xTrackExecute,

    // Gốc conveyor trong hệ robot/base.
    ConveyorBeltOrigin := stConveyorOriginSMC,

    // Pose object tại thời điểm tham chiếu ban đầu.
    InitialObjectPosition := stInitialObjectSMC,

    // Dùng PCS_1 cho ứng dụng Conveyor Tracking.
    CoordSystem := SMC_COORD_SYSTEM.PCS_1

);

//=============================================================================
// 04. CẬP NHẬT OUTPUT CHUNG
//=============================================================================

// Done của Manager là xung một chu kỳ.
Runtime.Response.Done := FALSE;

// SyncOK chỉ TRUE khi Robot đã tới Approach và PCS còn InUse.
SyncOK := FALSE;

// Released là xung một chu kỳ khi Multi-tool Core đã thoát PCS.
Released := FALSE;

// MotionRequest phản ánh trạng thái request nội bộ đang chờ Adapter nhận.
MotionRequest := xMotionRequestPending;

// TrackingActive TRUE khi Manager Busy, PCS Execute hoặc PCS đang InUse.
TrackingActive := Runtime.Response.Busy OR xTrackExecute OR fbTrackBelt.InUse;

// Đồng bộ trạng thái InUse của PCS vào Runtime.
Runtime.PCSInfo.InUse := fbTrackBelt.InUse;

//=============================================================================
// 05. RESET TOÀN BỘ MANAGER
//=============================================================================

IF Reset THEN
    // Đưa state machine về IDLE.
    Runtime.State := E_TrackingState.TRK_IDLE;

    // Xóa phản hồi Accepted.
    Runtime.Response.Accepted := FALSE;

    // Xóa phản hồi Busy.
    Runtime.Response.Busy := FALSE;

    // Xóa phản hồi Done.
    Runtime.Response.Done := FALSE;

    // Xóa phản hồi Error.
    Runtime.Response.Error := FALSE;

    // Xóa mã lỗi.
    Runtime.Response.ErrorID := 0;

    // Xóa index object active.
    Runtime.SelectedObjectIndex := 0;

    // Xóa ObjectID active.
    Runtime.SelectedObjectID := 0;

    // Xóa kết quả gắp.
    Runtime.PickSuccess := FALSE;

    // Đánh dấu PCS chưa hợp lệ.
    Runtime.PCSInfo.Valid := FALSE;

    // Đánh dấu PCS không còn được sử dụng.
    Runtime.PCSInfo.InUse := FALSE;

    // Hạ Execute của MC_TrackConveyorBelt.
    xTrackExecute := FALSE;

    // Xóa cờ đã phát motion.
    xMotionIssued := FALSE;

    // Xóa request motion đang chờ.
    xMotionRequestPending := FALSE;

    // Xóa trạng thái motion active.
    xMotionActive := FALSE;

    // Xóa trạng thái đã hút được vật.
    xVacuumCaptured := FALSE;

    // Tắt yêu cầu van hút.
    VacuumCommand := FALSE;

    // Tắt yêu cầu van thổi.
    BlowCommand := FALSE;

    // Hạ yêu cầu abort motion.
    MotionAbort := FALSE;

    // Xóa trạng thái đồng bộ và xung Release.
    SyncOK := FALSE;
    Released := FALSE;

    // Reset timer PickDelay.
    tonPickDelay(IN := FALSE);

    // Reset timer VacuumTimeout.
    tonVacuumTimeout(IN := FALSE);

    // Reset timer Blow.
    tonBlow(IN := FALSE);
	
	stToolSyncPos.X := 0.0;
	stToolSyncPos.Y := 0.0;
	stToolSyncPos.Z := 0.0;
	stToolSyncPos.A := 0.0;
	xPickPositionReady := FALSE;
	xPickMotionBusySeen := FALSE;
	xRetractMotionBusySeen := FALSE;
    // Kết thúc xử lý trong cycle reset.
	
	xPCSStartCaptured := FALSE;
	lrConveyorPosAtPCSStart := 0.0;
	lrDeltaCaptureToPCS := 0.0;

    RETURN;
END_IF;

//=============================================================================
// 06. HẠ EXECUTE KHI MANAGER ĐANG BUSY -> ABORT CÓ KIỂM SOÁT
//=============================================================================

//=============================================================================
// EXECUTE BỊ HẠ TRONG KHI MANAGER CHƯA KẾT THÚC
//=============================================================================
//=============================================================================
// EXECUTE ĐÃ HẠ - KHÔNG CHO STATE MACHINE TIẾP TỤC REQUEST CŨ
//=============================================================================

IF NOT Execute
AND Runtime.State <> E_TrackingState.TRK_IDLE
AND Runtime.State <> E_TrackingState.TRK_COMPLETE
AND Runtime.State <> E_TrackingState.TRK_ABORTING
AND Runtime.State <> E_TrackingState.TRK_ERROR THEN
    Runtime.State := E_TrackingState.TRK_ABORTING;
END_IF;


//=============================================================================
// 07. STATE MACHINE CHÍNH
//=============================================================================

CASE Runtime.State OF

    //=========================================================================
    // TRK_IDLE
    // Chờ lệnh Execute từ Application Manager hoặc chương trình test.
    //=========================================================================
    E_TrackingState.TRK_IDLE:

        // Manager chưa tiếp nhận lệnh.
        Runtime.Response.Accepted := FALSE;

        // Manager không bận.
        Runtime.Response.Busy := FALSE;

        // Xóa lỗi cũ khi về IDLE.
        Runtime.Response.Error := FALSE;

        // Xóa mã lỗi cũ.
        Runtime.Response.ErrorID := 0;

        // Không có object active.
        Runtime.SelectedObjectIndex := 0;

        // Không có ObjectID active.
        Runtime.SelectedObjectID := 0;

        // Xóa trạng thái gắp.
        Runtime.PickSuccess := FALSE;

        // Tắt hút.
        VacuumCommand := FALSE;

        // Tắt thổi.
        BlowCommand := FALSE;

        // Hạ abort motion.
        MotionAbort := FALSE;

        // Xóa cờ motion.
        xMotionIssued := FALSE;
        xMotionRequestPending := FALSE;
        xMotionActive := FALSE;

        // Xóa trạng thái tool đã giữ vật.
        xVacuumCaptured := FALSE;

        // Khi Execute TRUE, tiếp nhận lệnh và bắt đầu tìm object.
        IF Execute THEN
            // Báo đã tiếp nhận request.
            Runtime.Response.Accepted := TRUE;

            // Báo Manager đang bận.
            Runtime.Response.Busy := TRUE;

            // Chuyển sang Scheduler.
            Runtime.State := E_TrackingState.TRK_FIND_OBJECT;
        END_IF;

//     //=========================================================================
//     // TRK_FIND_OBJECT
//     // Scheduler tìm object phù hợp nhất trong Queue.
//     //=========================================================================
    E_TrackingState.TRK_FIND_OBJECT:

        VacuumCommand := FALSE;
        BlowCommand := FALSE;

        IF UseExternalSelection THEN
            IF ExternalObjectIndex = 0 THEN
				Runtime.Response.Error := FALSE;
				Runtime.Response.ErrorID := 0;
			
			ELSIF ExternalObjectIndex > GVL.C_MAX_TRACK_OBJECTS THEN
				Runtime.Response.Error := TRUE;
				Runtime.Response.ErrorID := 6501;
				Runtime.State := E_TrackingState.TRK_ERROR;
                
            ELSIF NOT Queue.Objects[ExternalObjectIndex].Valid THEN
                Runtime.Response.Error := TRUE;
                Runtime.Response.ErrorID := 6502;
                Runtime.State := E_TrackingState.TRK_ERROR;
            ELSE
                Runtime.SelectedObjectIndex := ExternalObjectIndex;
                Runtime.SelectedObjectID := Queue.Objects[ExternalObjectIndex].ObjectID;
                Runtime.State := E_TrackingState.TRK_RESERVE_OBJECT;
            END_IF;

        ELSIF TestFixedObjectMode THEN
            Runtime.SelectedObjectIndex := 1;
            Runtime.SelectedObjectID := 1;
            Queue.Objects[1].Valid := TRUE;
            Queue.Objects[1].ObjectID := 1;
            Queue.Objects[1].Reserved := FALSE;
            Queue.Objects[1].CanPick := TRUE;
            Queue.Objects[1].AbortRequired := FALSE;
            Queue.Objects[1].State := E_TrackingObjectState.OBJ_READY;
            Runtime.State := E_TrackingState.TRK_RESERVE_OBJECT;

        ELSE
            uiSelectedIndex := F_SelectTrackingObject(
                SelectMode := Config.SelectMode,
                SpecificID := Config.SpecificObjectID,
                DirectionSign := ConveyorConfig.DirectionSign,
                MinimumVisionScore := Config.MinimumVisionScore,
                Queue := Queue
            );

            IF uiSelectedIndex <> GVL.C_INVALID_INDEX THEN
                Runtime.SelectedObjectIndex := uiSelectedIndex;
                Runtime.SelectedObjectID := Queue.Objects[uiSelectedIndex].ObjectID;
                Runtime.State := E_TrackingState.TRK_RESERVE_OBJECT;
            END_IF;
        END_IF;


    //=========================================================================
    // TRK_RESERVE_OBJECT
    // Kiểm tra object lần cuối rồi khóa quyền sở hữu.
    //=========================================================================
    E_TrackingState.TRK_RESERVE_OBJECT:

        // Nếu index không hợp lệ thì quay lại tìm object.
        IF Runtime.SelectedObjectIndex = GVL.C_INVALID_INDEX THEN
            Runtime.State := E_TrackingState.TRK_FIND_OBJECT;

        // Nếu slot không còn hợp lệ thì hủy lựa chọn.
        ELSIF NOT Queue.Objects[Runtime.SelectedObjectIndex].Valid THEN

            Runtime.SelectedObjectIndex := 0;
            Runtime.SelectedObjectID := 0;

            Runtime.State := E_TrackingState.TRK_FIND_OBJECT;

        // Nếu object đã bị module khác Reserve thì báo lỗi tranh chấp.
        ELSIF Queue.Objects[Runtime.SelectedObjectIndex].Reserved THEN

            Runtime.Response.Error := TRUE;
            Runtime.Response.ErrorID := 6001;

            Runtime.State := E_TrackingState.TRK_ERROR;

        // Nếu object không còn đủ điều kiện gắp thì đánh dấu MISSED.
        ELSIF NOT Queue.Objects[Runtime.SelectedObjectIndex].CanPick THEN

            Queue.Objects[Runtime.SelectedObjectIndex].State := E_TrackingObjectState.OBJ_MISSED;

            // MissCode 1: mất điều kiện trước khi Reserve.
            Queue.Objects[Runtime.SelectedObjectIndex].MissCode := 1;

            Queue.Objects[Runtime.SelectedObjectIndex].Reserved := FALSE;

            Runtime.SelectedObjectIndex := 0;
            Runtime.SelectedObjectID := 0;

            Runtime.State := E_TrackingState.TRK_FIND_OBJECT;

        ELSE
            // Khóa object cho Manager này.
            Queue.Objects[Runtime.SelectedObjectIndex].Reserved := TRUE;

            // Chuyển trạng thái object sang RESERVED.
            Queue.Objects[Runtime.SelectedObjectIndex].State := E_TrackingObjectState.OBJ_RESERVED;

            // Ghi ActiveIndex vào Queue.
            Queue.ActiveIndex := Runtime.SelectedObjectIndex;

            // Xóa trạng thái hút cũ.
            xVacuumCaptured := FALSE;

            // Xóa kết quả gắp cũ.
            Runtime.PickSuccess := FALSE;

            // Chuyển sang kiểm tra vùng gắp.
            Runtime.State := E_TrackingState.TRK_WAIT_PICK_ZONE;
        END_IF;

    //=========================================================================
    // TRK_WAIT_PICK_ZONE
    // Chờ object còn nằm trong vùng an toàn và đủ thời gian.
    //=========================================================================
    E_TrackingState.TRK_WAIT_PICK_ZONE:

        // Nếu object mất hiệu lực thì giải phóng.
        IF NOT Queue.Objects[Runtime.SelectedObjectIndex].Valid THEN

            Runtime.State := E_TrackingState.TRK_RELEASE_OBJECT;

        // Nếu object đã qua mốc Abort trước khi tạo PCS.
        ELSIF Queue.Objects[Runtime.SelectedObjectIndex].AbortRequired THEN

            Queue.Objects[Runtime.SelectedObjectIndex].State := E_TrackingObjectState.OBJ_MISSED;

            // MissCode 2: quá vùng trong WAIT_PICK_ZONE.
            Queue.Objects[Runtime.SelectedObjectIndex].MissCode := 2;

            Runtime.State := E_TrackingState.TRK_RELEASE_OBJECT;

        // Nếu object còn đủ điều kiện gắp thì chuẩn bị PCS.
        ELSIF Queue.Objects[Runtime.SelectedObjectIndex].CanPick THEN

            Runtime.State := E_TrackingState.TRK_PREPARE_PCS;
        END_IF;

    //=========================================================================
    // TRK_PREPARE_PCS
    // Chụp dữ liệu object active và tạo các điểm trong PCS.
    //=========================================================================
    E_TrackingState.TRK_PREPARE_PCS:

        // Sao chép object active để tránh đọc rời rạc nhiều lần.
        stSelectedObject := Queue.Objects[Runtime.SelectedObjectIndex];

        // Lưu ObjectID vào thông tin PCS.
        Runtime.PCSInfo.ObjectID := stSelectedObject.ObjectID;

        //=========================================================================
        // CHỌN NGUỒN VỊ TRÍ OBJECT
        //-------------------------------------------------------------------------
        // Trong chế độ test:
        //     dùng vị trí object cố định.
        //
        // Trong chế độ chạy thật:
		//     dùng Pose chuẩn của Object trong Queue.
		//     Sensor/Vision đều phải chuẩn hóa về PoseInConveyor.
        //=========================================================================
        IF TestFixedObjectMode THEN
        
            // Gán vị trí object test cố định.
            Runtime.PCSInfo.InitialObjectPos.X := FixedObjectPosition.X;
        
            Runtime.PCSInfo.InitialObjectPos.Y := FixedObjectPosition.Y;
        
            Runtime.PCSInfo.InitialObjectPos.Z := FixedObjectPosition.Z;
        
            Runtime.PCSInfo.InitialObjectPos.A := FixedObjectPosition.A;
        

        
        ELSE			
			// Chế độ chạy thật lấy Pose chuẩn của Object trong hệ Conveyor.
			// Sensor/Vision đều phải chuẩn hóa dữ liệu vào PoseInConveyor
			// trước khi đưa Object vào Tracking Queue.
			
			
			Runtime.PCSInfo.InitialObjectPos := stSelectedObject.PoseInConveyor;
			
			//=============================================================
			// BÙ CHIỀU CAO MẶT HÚT SẢN PHẨM
			//=============================================================
			IF UseExternalSelection THEN
		
				Runtime.PCSInfo.InitialObjectPos.Z :=
					stSelectedObject.PoseInConveyor.Z
					+ ExternalPickSurfaceHeightMM;
		
			END_IF;
			
			
        END_IF;

        // Lưu gốc conveyor.
        //Runtime.PCSInfo.ConveyorOrigin := ConveyorOrigin;
        // Tọa độ X của gốc conveyor trong hệ robot/base.
        Runtime.PCSInfo.ConveyorOrigin.X := ConveyorOrigin.X;
        
        // Tọa độ Y của gốc conveyor trong hệ robot/base.
        Runtime.PCSInfo.ConveyorOrigin.Y := ConveyorOrigin.Y;
        
        // Tọa độ Z của gốc conveyor trong hệ robot/base.
        Runtime.PCSInfo.ConveyorOrigin.Z := ConveyorOrigin.Z;
        
        // Góc A của hệ conveyor.
        Runtime.PCSInfo.ConveyorOrigin.A := ConveyorOrigin.A;
    

        // Lưu vị trí conveyor tại thời điểm capture.
        //Runtime.PCSInfo.ConveyorCapturePos := stSelectedObject.CaptureConveyorPos;
		
		Runtime.PCSInfo.ConveyorCapturePos := LREAL_TO_REAL(stSelectedObject.CaptureConveyorPositionMM);
	
	
       // Quy ước:
		// - PickPos: điểm gắp thật của đầu Tool.
		// - ApproachPos: vị trí robot bắt đầu bám, phía trên PickPos.
		// - stToolSyncPos: cùng vị trí với ApproachPos.
		// - UseUpDown chỉ quyết định ai đi quãng cuối:
		//      TRUE  -> Tool cylinder đi xuống.
		//      FALSE -> Robot đi xuống.
		//=========================================================================
		IF UseExternalSelection THEN
		
			//---------------------------------------------------------------------
			// 1. ĐIỂM GẮP THẬT
			//---------------------------------------------------------------------
			Runtime.PickPos := ExternalPickOffset;
		
			//---------------------------------------------------------------------
			// 2. ĐIỂM ĐỒNG BỘ CỦA ROBOT
			// Luôn cao hơn điểm gắp bằng ApproachHeight,
			// không phụ thuộc Tool có Up/Down hay không.
			//---------------------------------------------------------------------
			Runtime.ApproachPos := Runtime.PickPos;
		
			Runtime.ApproachPos.Z := Runtime.PickPos.Z + ExternalApproachHeight;
		
			//---------------------------------------------------------------------
			// Robot bám conveyor tại chính điểm Approach.
			//---------------------------------------------------------------------
			stToolSyncPos := Runtime.ApproachPos;
		
			//---------------------------------------------------------------------
			// 3. ĐIỂM NÂNG SAU KHI GẮP
			// RetractHeight được tính từ điểm gắp thật.
			//---------------------------------------------------------------------
			Runtime.RetractPos := Runtime.PickPos;
		
			Runtime.RetractPos.Z := Runtime.PickPos.Z+ Config.RetractHeight;
		
		ELSE
		
			//---------------------------------------------------------------------
			// GIỮ LOGIC TRACKING THƯỜNG
			//---------------------------------------------------------------------
			Runtime.PickPos := Config.PickOffset;
		
			Runtime.ApproachPos := Config.PickOffset;
		
			Runtime.ApproachPos.Z :=
				Runtime.ApproachPos.Z
				+ Config.ApproachHeight;
		
			stToolSyncPos := Runtime.ApproachPos;
		
			Runtime.RetractPos := Config.PickOffset;
		
			Runtime.RetractPos.Z :=
				Runtime.RetractPos.Z
				+ Config.RetractHeight;
		
		END_IF;

	
		// Chu trình mới chưa tới vị trí sẵn sàng thao tác Tool.
		xPickPositionReady := FALSE;
		xPickMotionBusySeen := FALSE;
		xRetractMotionBusySeen := FALSE;
		xExitPCSTargetValid := FALSE;
        // PCS chưa hợp lệ trước khi SoftMotion báo Done.
        Runtime.PCSInfo.Valid := FALSE;
		
		// Cho phép PCS mới chụp lại Conveyor Position.
		// Mỗi Object mới vào TRK_PREPARE_PCS sẽ reset cờ này.
		xPCSStartCaptured := FALSE;

        // Chuyển sang tạo PCS.
        Runtime.State := E_TrackingState.TRK_CREATE_PCS;
		
		
	//=========================================================================
	// TRK_CREATE_PCS
	// Chốt vị trí Conveyor và tạo cạnh Execute cho MC_TrackConveyorBelt.
	//=========================================================================
	E_TrackingState.TRK_CREATE_PCS:
	
		//---------------------------------------------------------------------
		// CHỐT DỮ LIỆU PCS MỘT LẦN
		//---------------------------------------------------------------------
		IF NOT xPCSStartCaptured THEN
	
			// Vị trí Conveyor gần nhất trước lúc MC_TrackConveyorBelt Execute.
			lrConveyorPosAtPCSStart :=
				REAL_TO_LREAL(ConveyorStatus.PositionMM);
	
			// Conveyor đã dịch từ lúc Sensor/Vision Capture tới lúc tạo PCS.
			lrDeltaCaptureToPCS :=
				lrConveyorPosAtPCSStart
				- stSelectedObject.CaptureConveyorPositionMM;
	
			//-----------------------------------------------------------------
			// CẬP NHẬT POSE OBJECT TẠI THỜI ĐIỂM BẮT ĐẦU PCS
			//-----------------------------------------------------------------
			IF NOT TestFixedObjectMode THEN
	
// 				// PoseInConveyor là Pose tại thời điểm Capture.
// 				Runtime.PCSInfo.InitialObjectPos :=
// 					stSelectedObject.PoseInConveyor;
	
				// Conveyor chạy theo +X của Conveyor CS.
				Runtime.PCSInfo.InitialObjectPos.X :=
					stSelectedObject.PoseInConveyor.X
					+ LREAL_TO_REAL(lrDeltaCaptureToPCS);
	
			END_IF;
	
			// Đánh dấu đã chốt dữ liệu cho PCS hiện tại.
			xPCSStartCaptured := TRUE;
	
		END_IF;
	
		//---------------------------------------------------------------------
		// TẠO CẠNH EXECUTE CHO MC_TrackConveyorBelt
		//---------------------------------------------------------------------
		xTrackExecute := TRUE;
	
		// Sang state chờ SoftMotion tạo PCS.
		Runtime.State := E_TrackingState.TRK_WAIT_PCS;
	
	
	//=========================================================================
	// TRK_WAIT_PCS
	// Chờ MC_TrackConveyorBelt hoàn tất tạo PCS.
	//=========================================================================
	E_TrackingState.TRK_WAIT_PCS:
	
		// Quan trọng:
		// Giữ Execute TRUE trong toàn bộ vòng đời PCS.
		xTrackExecute := TRUE;
	
		//---------------------------------------------------------------------
		// TRACK CONVEYOR ERROR
		//---------------------------------------------------------------------
		IF fbTrackBelt.Error THEN
	
			Runtime.Response.Error := TRUE;
			Runtime.Response.ErrorID :=
				TO_UDINT(fbTrackBelt.ErrorID);
	
			Runtime.State :=
				E_TrackingState.TRK_ERROR;
	
		//---------------------------------------------------------------------
		// PCS ĐÃ ĐƯỢC TẠO
		//---------------------------------------------------------------------
		ELSIF fbTrackBelt.Done THEN
	
			// Không hạ xTrackExecute ở đây.
			Runtime.PCSInfo.Valid := TRUE;
	
			// Đánh dấu Object đã có Dynamic PCS.
			Queue.Objects[Runtime.SelectedObjectIndex].State :=
				E_TrackingObjectState.OBJ_PCS_READY;
	
			// Chuẩn bị phát Motion Approach.
			xMotionIssued := FALSE;
			xMotionRequestPending := FALSE;
			xMotionActive := FALSE;
	
			Runtime.State :=
				E_TrackingState.TRK_MOVE_APPROACH;
	
		END_IF;

//     //=========================================================================
//     // TRK_CREATE_PCS
//     // Tạo cạnh Execute cho MC_TrackConveyorBelt.
//     //=========================================================================
//     E_TrackingState.TRK_CREATE_PCS:
// 
//         // Bật Execute PCS.
//         xTrackExecute := TRUE;
// 
//         // Chuyển sang chờ SoftMotion tạo PCS.
//         Runtime.State := E_TrackingState.TRK_WAIT_PCS;
// 
//     //=========================================================================
//     // TRK_WAIT_PCS
//     // Chờ MC_TrackConveyorBelt hoàn tất tạo PCS.
//     //=========================================================================
//     E_TrackingState.TRK_WAIT_PCS:
// 
//         // Nếu SoftMotion báo lỗi.
//         IF fbTrackBelt.Error THEN
//             Runtime.Response.Error := TRUE;
// 
//             // Cast ErrorID theo kiểu Runtime đang sử dụng.
//             Runtime.Response.ErrorID := TO_UDINT(fbTrackBelt.ErrorID);
// 
//             Runtime.State := E_TrackingState.TRK_ERROR;
// 
//         // Khi PCS đã được tạo.
//         ELSIF fbTrackBelt.Done THEN
//             // Không hạ xTrackExecute tại đây.
//             Runtime.PCSInfo.Valid := TRUE;
// 
//             // Đánh dấu object đã có PCS.
//             Queue.Objects[Runtime.SelectedObjectIndex].State := E_TrackingObjectState.OBJ_PCS_READY;
// 
//             // Chuẩn bị phát motion Approach.
//             xMotionIssued := FALSE;
//             xMotionRequestPending := FALSE;
//             xMotionActive := FALSE;
// 
//             Runtime.State := E_TrackingState.TRK_MOVE_APPROACH;
//         END_IF;

    //=========================================================================
    // TRK_MOVE_APPROACH
    // Đi tới phía trên object trong PCS_1.
    //=========================================================================
    E_TrackingState.TRK_MOVE_APPROACH:

    // Trong chế độ test cố định, không cho Updater abort object test.
    IF TestFixedObjectMode THEN
        Queue.Objects[Runtime.SelectedObjectIndex].AbortRequired := FALSE;
    END_IF;

    // Chỉ tạo một request mới khi chưa có request/motion nào active.
    IF NOT xMotionIssued AND NOT xMotionRequestPending AND NOT xMotionActive THEN

        // Điểm đích Approach trong PCS_1.
        MotionTarget := Runtime.ApproachPos;

        // Tốc độ Approach lấy từ Tracking Config.
        MotionSpeed := Config.Motion.Approach.Speed;

        // Gia tốc Approach.
        MotionAcceleration := Config.Motion.Approach.Acceleration;

        // Giảm tốc Approach.
        MotionDeceleration := Config.Motion.Approach.Deceleration;

        // Jerk Approach.
        MotionJerk := Config.Motion.Approach.Jerk;

        // Blend radius của Approach.
        MotionBlendRadius := Config.Motion.Approach.BlendRadius;

        // Approach được thực hiện trong PCS động số 1.
        MotionCoordSystem := E_AppCoordSystem.APP_COORD_PCS1;

        // Mã lệnh MoveL.
        MotionCommand := 2;

        // Chỉ phát request nếu dữ liệu motion hợp lệ.
        IF MotionSpeed > 0.0 AND MotionAcceleration > 0.0 AND MotionDeceleration > 0.0 THEN

            // Đánh dấu request đang chờ Motion Adapter nhận.
            xMotionRequestPending := TRUE;

            // Đánh dấu state đã tạo request.
            xMotionIssued := TRUE;

        ELSE
            // Thông số Dynamic bằng 0 nên không được phát motion.
            Runtime.Response.Error := TRUE;

            // Mã lỗi nội bộ: cấu hình Approach không hợp lệ.
            Runtime.Response.ErrorID := 6101;

            // Chuyển sang state lỗi.
            Runtime.State := E_TrackingState.TRK_ERROR;
        END_IF;
    END_IF;

    // Motion Adapter đã nhận request.
    IF MotionAccepted AND xMotionRequestPending THEN

        // Hạ request pending.
        xMotionRequestPending := FALSE;

        // Bắt đầu chờ MotionDone.
        xMotionActive := TRUE;
    END_IF;

    // Motion Approach hoàn thành.
    IF MotionDone AND xMotionActive THEN
		xMotionActive := FALSE;
		xMotionIssued := FALSE;
		xMotionRequestPending := FALSE;
	
		IF UseExternalSelection THEN
			IF ExternalUseUpDown THEN
				// Robot đã tới SyncPos.
				// Tool cơ khí sẽ thực hiện hành trình xuống.
				xPickPositionReady := TRUE;
			ELSE
				// Robot mới chỉ tới SyncPos.
				// Bắt buộc phải phát thêm MoveL xuống PickPos.
				xPickPositionReady := FALSE;
			END_IF;
		ELSE
			xPickPositionReady := FALSE;
		END_IF;
	
		Runtime.State := E_TrackingState.TRK_MOVE_PICK;
	
	ELSIF MotionError AND xMotionActive THEN
		xMotionActive := FALSE;
		xMotionIssued := FALSE;
		xMotionRequestPending := FALSE;
	
		Runtime.Response.Error := TRUE;
		Runtime.Response.ErrorID := MotionErrorID;
		Runtime.State := E_TrackingState.TRK_ERROR;
	END_IF;

    //=========================================================================
    // TRK_MOVE_PICK
    // Hạ TCP từ Approach xuống PickPos trong PCS_1.
    //=========================================================================
    E_TrackingState.TRK_MOVE_PICK:

        IF UseExternalSelection THEN
            xTrackExecute := TRUE;
			VacuumCommand := FALSE;
			BlowCommand := FALSE;
	
			//---------------------------------------------------------------------
			// Chưa tới vị trí sẵn sàng thì phát một MoveL trong PCS_1.
			//---------------------------------------------------------------------
			IF NOT xPickPositionReady THEN

				IF NOT xMotionIssued AND NOT xMotionRequestPending AND NOT xMotionActive THEN
			
					Queue.Objects[Runtime.SelectedObjectIndex].State := E_TrackingObjectState.OBJ_PICKING;
			
					// Không có Up/Down:
					// robot phải tự xuống điểm Pick thật.
					MotionTarget := Runtime.PickPos;
			
					MotionSpeed := Config.Motion.Pick.Speed;
					MotionAcceleration := Config.Motion.Pick.Acceleration;
					MotionDeceleration := Config.Motion.Pick.Deceleration;
					MotionJerk := Config.Motion.Pick.Jerk;
					MotionBlendRadius := Config.Motion.Pick.BlendRadius;
					MotionCoordSystem := E_AppCoordSystem.APP_COORD_PCS1;
					MotionCommand := 2;
			
					xPickMotionBusySeen := FALSE;
					xMotionRequestPending := TRUE;
					xMotionIssued := TRUE;
				END_IF;
			
				IF MotionAccepted AND xMotionRequestPending THEN
					xMotionRequestPending := FALSE;
					xMotionActive := TRUE;
				END_IF;
			
				IF xMotionActive AND MotionBusy THEN
					xPickMotionBusySeen := TRUE;
				END_IF;
			
				IF MotionDone
				AND xMotionActive
				AND xPickMotionBusySeen THEN
			
					xMotionActive := FALSE;
					xMotionIssued := FALSE;
					xMotionRequestPending := FALSE;
					xPickMotionBusySeen := FALSE;
			
					// Chỉ tới đây mới xác nhận robot đã xuống PickPos.
					xPickPositionReady := TRUE;
			
				ELSIF MotionError AND xMotionActive THEN
			
					xMotionActive := FALSE;
					xMotionIssued := FALSE;
					xMotionRequestPending := FALSE;
					xPickMotionBusySeen := FALSE;
			
					Runtime.Response.Error := TRUE;
					Runtime.Response.ErrorID := MotionErrorID;
					Runtime.State := E_TrackingState.TRK_ERROR;
				END_IF;
			
			END_IF;
	
			//---------------------------------------------------------------------
			// Chỉ báo SyncOK sau khi robot tới đúng vị trí thao tác.
			//---------------------------------------------------------------------
			SyncOK := xPickPositionReady AND Runtime.PCSInfo.Valid AND fbTrackBelt.InUse;
	
			//---------------------------------------------------------------------
			// Controller đã hoàn thành:
			// - Có Up/Down: DOWN -> GRIP -> UP.
			// - Không Up/Down: GRIP.
			//---------------------------------------------------------------------
			IF PickerSafe AND SyncOK THEN
	
				Runtime.PickSuccess := TRUE;
				xVacuumCaptured := TRUE;
				
				xRetractMotionBusySeen := FALSE;
				xExitPCSTargetValid := FALSE;
				
				IF ExternalUseUpDown THEN
					// Tool đã thực hiện DOWN -> GRIP -> UP.
					// Robot vẫn đang tại Sync/ApproachPos.
					// Không được chạy xuống RetractPos.
					Runtime.State := E_TrackingState.TRK_LEAVE_PCS;
				ELSE
					// Không có Tool Up/Down.
					// Robot đang tại PickPos và cần tự nâng lên RetractPos.
					Runtime.State := E_TrackingState.TRK_MOVE_RETRACT;
				END_IF;
					
			ELSIF fbTrackBelt.Error THEN
	
				Runtime.Response.Error := TRUE;
				Runtime.Response.ErrorID :=
					TO_UDINT(fbTrackBelt.ErrorID);
				Runtime.State := E_TrackingState.TRK_ERROR;
	
			END_IF;

        ELSE


            // Chưa VacuumOK nên vẫn có thể abort nếu object quá vùng.
            IF Queue.Objects[Runtime.SelectedObjectIndex].AbortRequired AND NOT xVacuumCaptured THEN

                Queue.Objects[Runtime.SelectedObjectIndex].State := E_TrackingObjectState.OBJ_MISSED;

                // MissCode 4: quá vùng trong Move Pick.
                Queue.Objects[Runtime.SelectedObjectIndex].MissCode := 4;

                MotionAbort := TRUE;

                Runtime.State := E_TrackingState.TRK_ABORT_ACTIVE;

            ELSE
                // Tạo request Pick mới.
                IF NOT xMotionIssued AND NOT xMotionRequestPending AND NOT xMotionActive THEN

                    // Đánh dấu object đang ở pha Picking.
                    Queue.Objects[Runtime.SelectedObjectIndex].State := E_TrackingObjectState.OBJ_PICKING;

                    // Gán điểm Pick.
                    MotionTarget := Runtime.PickPos;

                    // Gán tốc độ Pick.
                    MotionSpeed := Config.Motion.Pick.Speed;

                    // Gán gia tốc Pick.
                    MotionAcceleration := Config.Motion.Pick.Acceleration;

                    // Gán giảm tốc Pick.
                    MotionDeceleration := Config.Motion.Pick.Deceleration;

                    // Gán jerk Pick.
                    MotionJerk := Config.Motion.Pick.Jerk;

                    // Gán blend Pick.
                    MotionBlendRadius := Config.Motion.Pick.BlendRadius;

                    // Pick chạy trong PCS_1.
                    MotionCoordSystem := E_AppCoordSystem.APP_COORD_PCS1;

                    // Mã lệnh MoveL.
                    MotionCommand := 2;

                    // Bật request pending.
                    xMotionRequestPending := TRUE;

                    // Đánh dấu đã tạo lệnh.
                    xMotionIssued := TRUE;
                END_IF;
					
					// Adapter đã nhận đúng request Pick.
					IF MotionAccepted AND xMotionRequestPending THEN
						xMotionRequestPending := FALSE;
						xMotionActive := TRUE;
					END_IF;
					
					// Phải thấy motion Pick thực sự Busy ít nhất một scan.
					// Nhờ đó không nhận nhầm Done còn lại từ lệnh Approach.
					IF xMotionActive AND MotionBusy THEN
						xPickMotionBusySeen := TRUE;
					END_IF;
					
					// Chỉ công nhận Done sau khi motion Pick đã thực sự Busy.
					IF MotionDone
					AND xMotionActive
					AND xPickMotionBusySeen THEN
					
						xMotionActive := FALSE;
						xMotionIssued := FALSE;
						xMotionRequestPending := FALSE;
						xPickMotionBusySeen := FALSE;
					
						xPickPositionReady := TRUE;
					
					ELSIF MotionError AND xMotionActive THEN
					
						xMotionActive := FALSE;
						xMotionIssued := FALSE;
						xMotionRequestPending := FALSE;
						xPickMotionBusySeen := FALSE;
					
						Runtime.Response.Error := TRUE;
						Runtime.Response.ErrorID := MotionErrorID;
						Runtime.State := E_TrackingState.TRK_ERROR;
					
					END_IF;

//                 // Adapter đã nhận request.
//                 IF MotionAccepted AND xMotionRequestPending THEN
//                     xMotionRequestPending := FALSE;
//                     xMotionActive := TRUE;
//                 END_IF;
// 
//                 // Motion Pick hoàn thành.
//                 IF MotionDone AND xMotionActive THEN
//                     xMotionActive := FALSE;
//                     xMotionIssued := FALSE;
// 
//                     Runtime.State := E_TrackingState.TRK_GRIP_ON;
// 
//                 // Motion Pick lỗi.
//                 ELSIF MotionError AND xMotionActive THEN
//                     xMotionActive := FALSE;
// 
//                     Runtime.Response.Error := TRUE;
//                     Runtime.Response.ErrorID := MotionErrorID;
// 
//                     Runtime.State := E_TrackingState.TRK_ERROR;
//                 END_IF;
            END_IF;

        END_IF;


    //=========================================================================
    // TRK_GRIP_ON
    // Bật hút và chờ PickDelay.
    //=========================================================================
    E_TrackingState.TRK_GRIP_ON:

        // Bật yêu cầu hút.
        VacuumCommand := TRUE;

        // Chạy timer PickDelay.
        tonPickDelay(
            IN := TRUE,
            PT := Config.PickDelay
        );

        // Khi hết thời gian chờ.
        IF tonPickDelay.Q THEN
            // Reset timer PickDelay.
            tonPickDelay(IN := FALSE);

            // Reset timer VacuumTimeout.
            tonVacuumTimeout(IN := FALSE);

            // Chuyển sang chờ VacuumOK.
            Runtime.State := E_TrackingState.TRK_WAIT_GRIP;
        END_IF;

    //=========================================================================
    // TRK_WAIT_GRIP
    // Chờ VacuumOK hoặc timeout.
    //=========================================================================
    E_TrackingState.TRK_WAIT_GRIP:

        // Giữ hút trong toàn bộ thời gian chờ.
        VacuumCommand := TRUE;

        // Chạy timer VacuumTimeout.
        tonVacuumTimeout(
            IN := TRUE,
            PT := Config.VacuumTimeout
        );

        // Nếu tool đã giữ được vật.
        IF VacuumOK THEN
            // Reset timeout.
            tonVacuumTimeout(IN := FALSE);

            // Khóa trạng thái đã hút thành công.
            xVacuumCaptured := TRUE;

            // Báo gắp thành công.
            Runtime.PickSuccess := TRUE;

            // Chuẩn bị phát motion Retract.
            xMotionIssued := FALSE;
            xMotionRequestPending := FALSE;
            xMotionActive := FALSE;

            Runtime.State := E_TrackingState.TRK_MOVE_RETRACT;

        // Nếu hết timeout mà chưa hút được.
        ELSIF tonVacuumTimeout.Q THEN
            // Reset timer.
            tonVacuumTimeout(IN := FALSE);

            // Tăng số lần thử.
            Queue.Objects[Runtime.SelectedObjectIndex].PickAttempts := Queue.Objects[Runtime.SelectedObjectIndex].PickAttempts + 1;

            // Nếu object đã vượt vùng an toàn thì không thử lại.
            IF Queue.Objects[Runtime.SelectedObjectIndex].AbortRequired THEN

                VacuumCommand := FALSE;

                Queue.Objects[Runtime.SelectedObjectIndex].State := E_TrackingObjectState.OBJ_MISSED;

                // MissCode 5: timeout và đã vượt vùng.
                Queue.Objects[Runtime.SelectedObjectIndex].MissCode := 5;

                Runtime.State := E_TrackingState.TRK_ABORT_ACTIVE;

            // Nếu còn lượt thử.
            ELSIF Queue.Objects[Runtime.SelectedObjectIndex].PickAttempts < Config.MaxPickAttempts THEN

                // Tắt hút trước lần thử tiếp theo.
                VacuumCommand := FALSE;

                // Cho phép phát lại lệnh Pick.
                xMotionIssued := FALSE;
                xMotionRequestPending := FALSE;
                xMotionActive := FALSE;

                Runtime.State := E_TrackingState.TRK_MOVE_PICK;

            ELSE
                // Hết số lần thử.
                VacuumCommand := FALSE;

                Queue.Objects[Runtime.SelectedObjectIndex].State := E_TrackingObjectState.OBJ_MISSED;

                // MissCode 6: hết số lần thử hút.
                Queue.Objects[Runtime.SelectedObjectIndex].MissCode := 6;

                Runtime.State := E_TrackingState.TRK_ABORT_ACTIVE;
            END_IF;
        END_IF;

    //=========================================================================
	// TRK_MOVE_RETRACT
	// Nâng sản phẩm trong PCS_1.
	//=========================================================================
	E_TrackingState.TRK_MOVE_RETRACT:
	
		// Giữ sản phẩm trong khi nâng.
		VacuumCommand := xVacuumCaptured;
		xTrackExecute := TRUE;
	
		//---------------------------------------------------------------------
		// PHÁT LỆNH RETRACT MỘT LẦN
		//---------------------------------------------------------------------
		IF NOT xMotionIssued
		AND NOT xMotionRequestPending
		AND NOT xMotionActive THEN
	
			// X/Y/A giữ nguyên theo PickPos; chỉ Z tăng.
			MotionTarget := Runtime.RetractPos;
	
			MotionSpeed := Config.Motion.Retract.Speed;
			MotionAcceleration := Config.Motion.Retract.Acceleration;
			MotionDeceleration := Config.Motion.Retract.Deceleration;
			MotionJerk := Config.Motion.Retract.Jerk;
			MotionBlendRadius := 0.0;
	
			// Vẫn bám vật trong lúc nâng.
			MotionCoordSystem := E_AppCoordSystem.APP_COORD_PCS1;
			MotionCommand := 2;
	
			xRetractMotionBusySeen := FALSE;
			xMotionRequestPending := TRUE;
			xMotionIssued := TRUE;
		END_IF;
	
		//---------------------------------------------------------------------
		// ADAPTER ĐÃ NHẬN LỆNH RETRACT
		//---------------------------------------------------------------------
		IF MotionAccepted AND xMotionRequestPending THEN
			xMotionRequestPending := FALSE;
			xMotionActive := TRUE;
		END_IF;
	
		//---------------------------------------------------------------------
		// CHÍNH LỆNH RETRACT ĐÃ THỰC SỰ CHẠY
		//---------------------------------------------------------------------
		IF xMotionActive AND MotionBusy THEN
			xRetractMotionBusySeen := TRUE;
		END_IF;
	
		//---------------------------------------------------------------------
		// RETRACT HOÀN THÀNH THẬT
		//---------------------------------------------------------------------
		IF MotionDone
		AND xMotionActive
		AND xRetractMotionBusySeen THEN
	
			xMotionActive := FALSE;
			xMotionIssued := FALSE;
			xMotionRequestPending := FALSE;
			xRetractMotionBusySeen := FALSE;
		
			xExitPCSTargetValid := FALSE;
		
			Runtime.State := E_TrackingState.TRK_LEAVE_PCS;
// 			xMotionActive := FALSE;
// 			xMotionIssued := FALSE;
// 			xMotionRequestPending := FALSE;
// 			xRetractMotionBusySeen := FALSE;
// 	
// 			xExitPCSTargetValid := FALSE;
// 	
// 			//-----------------------------------------------------------------
// 			// Chỉ sau khi nâng xong mới chụp vị trí MCS hiện tại.
// 			//-----------------------------------------------------------------
// 			stExitPCSTarget.X :=
// 				TO_REAL(POU_MONITOR_ROBOT.RB1_POS.c.X);
// 	
// 			stExitPCSTarget.Y :=
// 				TO_REAL(POU_MONITOR_ROBOT.RB1_POS.c.Y);
// 	
// 			stExitPCSTarget.Z :=
// 				TO_REAL(POU_MONITOR_ROBOT.RB1_POS.c.Z);
// 	
// 			stExitPCSTarget.A :=
// 				TO_REAL(POU_MONITOR_ROBOT.RB1_POS.c.A);
// 	
// 			// Chỉ cộng thêm Z, không thay đổi X/Y/A.
// 			stExitPCSTarget.Z :=
// 				stExitPCSTarget.Z + rExitPCSOffsetZ;
// 	
// 			IF stExitPCSTarget.Z < 0.0
// 			OR stExitPCSTarget.Z > rExitPCSMaxZ THEN
// 	
// 				Runtime.Response.Error := TRUE;
// 				Runtime.Response.ErrorID := 6130;
// 				Runtime.State := E_TrackingState.TRK_ERROR;
// 	
// 			ELSE
// 	
// 				xExitPCSTargetValid := TRUE;
// 				Runtime.State := E_TrackingState.TRK_LEAVE_PCS;
// 	
// 			END_IF;
	
		ELSIF MotionError AND xMotionActive THEN
	
			xMotionActive := FALSE;
			xMotionIssued := FALSE;
			xMotionRequestPending := FALSE;
			xRetractMotionBusySeen := FALSE;
	
			Runtime.Response.Error := TRUE;
			Runtime.Response.ErrorID := MotionErrorID;
			Runtime.State := E_TrackingState.TRK_ERROR;
	
		END_IF;


	//=============================================================================
	// TRK_LEAVE_PCS — STATE 120
	//-----------------------------------------------------------------------------
	// Phát một motion ngắn trong Robot Base/MCS để AxisGroup rời PCS_1.
	//
	// stExitPCSTarget đã được chụp một lần tại cuối Retract.
	// Không cập nhật stExitPCSTarget trong state này.
	//=============================================================================
	E_TrackingState.TRK_LEAVE_PCS:
	
		// Tiếp tục giữ sản phẩm.
		VacuumCommand := xVacuumCaptured;
	
		// Giữ MC_TrackConveyorBelt hoạt động cho tới khi AxisGroup rời PCS.
		xTrackExecute := TRUE;
	
		//---------------------------------------------------------------------
		// CHỤP TARGET MCS VÀ PHÁT MOTION EXIT PCS MỘT LẦN
		//---------------------------------------------------------------------
		IF NOT xMotionIssued
		AND NOT xMotionRequestPending
		AND NOT xMotionActive THEN
	
			// Chụp vị trí MCS muộn nhất có thể,
			// ngay trước khi tạo request Motion Queue.
// 			stExitPCSTarget.X :=
// 				TO_REAL(POU_MONITOR_ROBOT.RB1_POS.c.X);
// 	
// 			stExitPCSTarget.Y :=
// 				TO_REAL(POU_MONITOR_ROBOT.RB1_POS.c.Y);
// 	
// 			stExitPCSTarget.Z :=
// 				TO_REAL(POU_MONITOR_ROBOT.RB1_POS.c.Z);
// 	
// 			stExitPCSTarget.A :=
// 				TO_REAL(POU_MONITOR_ROBOT.RB1_POS.c.A);

			stExitPCSTarget.X :=
				TO_REAL(POU_COORDINATE_.Pos_Out_A_MCS.c.X);
	
			stExitPCSTarget.Y :=
				TO_REAL(POU_COORDINATE_.Pos_Out_A_MCS.c.Y);
	
			stExitPCSTarget.Z :=
				TO_REAL(POU_COORDINATE_.Pos_Out_A_MCS.c.Z);
	
			stExitPCSTarget.A :=
				TO_REAL(POU_COORDINATE_.Pos_Out_A_MCS.c.A);
	
			// Chỉ nâng thêm Z; không cộng offset X/Y/A.
			stExitPCSTarget.X := stExitPCSTarget.X - rExitPCSOffsetX;
			stExitPCSTarget.Z := stExitPCSTarget.Z + rExitPCSOffsetZ;
	
			//-----------------------------------------------------------------
			// KIỂM TRA TARGET
			//-----------------------------------------------------------------
			IF stExitPCSTarget.Z < 0.0
			OR stExitPCSTarget.Z > rExitPCSMaxZ THEN
	
				Runtime.Response.Error := TRUE;
				Runtime.Response.ErrorID := 6130;
				Runtime.State := E_TrackingState.TRK_ERROR;
	
			ELSE
	
				xExitPCSTargetValid := TRUE;
	
				MotionTarget := stExitPCSTarget;
	
				MotionSpeed := 80.0;
				MotionAcceleration := 300.0;
				MotionDeceleration := 300.0;
				MotionJerk := 1000.0;
				MotionBlendRadius := 0.0;
	
				// Chạy trong Robot Base/MCS để thoát khỏi PCS_1.
				MotionCoordSystem :=
					E_AppCoordSystem.APP_COORD_ROBOT_BASE;
	
				MotionCommand := 2;
	
				xMotionRequestPending := TRUE;
				xMotionIssued := TRUE;
	
			END_IF;
	
		END_IF;
	
		//---------------------------------------------------------------------
		// ADAPTER ĐÃ NHẬN MOTION EXIT PCS
		//---------------------------------------------------------------------
		IF MotionAccepted AND xMotionRequestPending THEN
			xMotionRequestPending := FALSE;
			xMotionActive := TRUE;
		END_IF;
	
		//---------------------------------------------------------------------
		// EXIT PCS HOÀN THÀNH
		//---------------------------------------------------------------------
		IF MotionDone AND xMotionActive THEN
	
			xMotionActive := FALSE;
			xMotionIssued := FALSE;
			xMotionRequestPending := FALSE;
	
			Runtime.State := E_TrackingState.TRK_RELEASE_PCS;
	
		ELSIF MotionError AND xMotionActive THEN
	
			xMotionActive := FALSE;
			xMotionIssued := FALSE;
			xMotionRequestPending := FALSE;
	
			Runtime.Response.Error := TRUE;
			Runtime.Response.ErrorID := MotionErrorID;
			Runtime.State := E_TrackingState.TRK_ERROR;
	
		END_IF;


	//=============================================================================
	// TRK_RELEASE_PCS — STATE 130
	//-----------------------------------------------------------------------------
	// Motion Exit PCS trong MCS đã hoàn thành.
	// Chờ SoftMotion xác nhận PCS_1 không còn được AxisGroup sử dụng.
	//=============================================================================
	E_TrackingState.TRK_RELEASE_PCS:
	
		// Tiếp tục giữ sản phẩm.
		VacuumCommand := xVacuumCaptured;
	
		// Không còn motion pending.
		xMotionIssued := FALSE;
		xMotionRequestPending := FALSE;
		xMotionActive := FALSE;
	
		// Trong lúc InUse vẫn TRUE, giữ FB Track còn Execute.
		xTrackExecute := TRUE;
	
		//---------------------------------------------------------------------
		// AXIS GROUP ĐÃ RỜI PCS_1
		//---------------------------------------------------------------------
		IF NOT fbTrackBelt.InUse THEN
	
			// Bây giờ mới được hạ Execute của MC_TrackConveyorBelt.
			xTrackExecute := FALSE;
	
			Runtime.PCSInfo.Valid := FALSE;
			Runtime.PCSInfo.InUse := FALSE;
	
			xExitPCSTargetValid := FALSE;
	
			IF UseExternalSelection THEN
                Released := TRUE;
                Runtime.Response.Done := TRUE;
                Runtime.Response.Busy := FALSE;
                Runtime.State := E_TrackingState.TRK_COMPLETE;
            ELSE
                Runtime.State := E_TrackingState.TRK_MOVE_SAFE_LEAVE;
            END_IF;
	
		//---------------------------------------------------------------------
		// TRACK CONVEYOR BÁO LỖI
		//---------------------------------------------------------------------
		ELSIF fbTrackBelt.Error THEN
	
			Runtime.Response.Error := TRUE;
			Runtime.Response.ErrorID := fbTrackBelt.ErrorID;
			Runtime.State := E_TrackingState.TRK_ERROR;
		END_IF;
	
	//=============================================================================
	// TRK_MOVE_SAFE_LEAVE
	//-----------------------------------------------------------------------------
	// PCS đã được release hoàn toàn.
	// Robot thực hiện MoveL tới điểm an toàn tuyệt đối trong Robot Base.
	//
	// Config.LeavePos phải là một điểm đã được dạy và test bằng Jog/MoveL riêng.
	// Không tính bằng cách cộng offset từ TCP hiện tại.
	//=============================================================================
	E_TrackingState.TRK_MOVE_SAFE_LEAVE:
	
		// Tiếp tục giữ sản phẩm.
		VacuumCommand := xVacuumCaptured;
	
		// Không cho MC_TrackConveyorBelt hoạt động lại.
		xTrackExecute := FALSE;
	
		// Tạo request motion một lần.
		IF NOT xMotionIssued
		AND NOT xMotionRequestPending
		AND NOT xMotionActive THEN
	
			// Điểm an toàn tuyệt đối trong Robot Base.
			MotionTarget := Config.LeavePos;
	
			// Thông số chuyển động Leave.
			MotionSpeed := Config.Motion.Leave.Speed;
			MotionAcceleration := Config.Motion.Leave.Acceleration;
			MotionDeceleration := Config.Motion.Leave.Deceleration;
			MotionJerk := Config.Motion.Leave.Jerk;
	
			// Không blend tại bước chuyển hệ tọa độ.
			MotionBlendRadius := 0.0;
	
			// Motion chạy trong Robot Base/MCS.
			MotionCoordSystem := E_AppCoordSystem.APP_COORD_ROBOT_BASE;
	
			// MoveL.
			MotionCommand := 2;
	
			// Phát yêu cầu tới Motion Adapter.
			xMotionRequestPending := TRUE;
			xMotionIssued := TRUE;
	
		END_IF;
	
		// Motion Adapter đã nhận lệnh.
		IF MotionAccepted AND xMotionRequestPending THEN
			xMotionRequestPending := FALSE;
			xMotionActive := TRUE;
		END_IF;
	
		// Điểm Safe Leave hoàn thành.
		IF MotionDone AND xMotionActive THEN
	
			xMotionActive := FALSE;
			xMotionIssued := FALSE;
			xMotionRequestPending := FALSE;
	
			Runtime.State := E_TrackingState.TRK_MOVE_PLACE;
	
		// Motion Safe Leave báo lỗi.
		ELSIF MotionError AND xMotionActive THEN
	
			xMotionActive := FALSE;
			xMotionIssued := FALSE;
			xMotionRequestPending := FALSE;
	
			Runtime.Response.Error := TRUE;
			Runtime.Response.ErrorID := MotionErrorID;
	
			Runtime.State := E_TrackingState.TRK_ERROR;
	
		END_IF;
		

    //=========================================================================
    // TRK_MOVE_PLACE
    // Di chuyển từ LeavePos tới PlacePos trong hệ robot/base.
    //=========================================================================
    E_TrackingState.TRK_MOVE_PLACE:

        // Giữ hút tới khi tới điểm đặt.
        VacuumCommand := xVacuumCaptured;

        // Tạo request Place mới.
        IF NOT xMotionIssued AND NOT xMotionRequestPending AND NOT xMotionActive THEN

            // Gán điểm Place.
            MotionTarget := Config.PlacePos;

            // Gán tốc độ Place.
            MotionSpeed := Config.Motion.Place.Speed;

            // Gán gia tốc Place.
            MotionAcceleration := Config.Motion.Place.Acceleration;

            // Gán giảm tốc Place.
            MotionDeceleration := Config.Motion.Place.Deceleration;

            // Gán jerk Place.
            MotionJerk := Config.Motion.Place.Jerk;

            // Gán blend Place.
            MotionBlendRadius := Config.Motion.Place.BlendRadius;

            // Place chạy trong hệ robot/base.
            MotionCoordSystem := E_AppCoordSystem.APP_COORD_ROBOT_BASE;

            // Mã lệnh MoveL.
            MotionCommand := 2;

            // Bật request pending.
            xMotionRequestPending := TRUE;

            // Đánh dấu đã tạo lệnh.
            xMotionIssued := TRUE;
        END_IF;

        // Adapter đã nhận request.
        IF MotionAccepted AND xMotionRequestPending THEN
            xMotionRequestPending := FALSE;
            xMotionActive := TRUE;
        END_IF;

        // Place hoàn thành.
        IF MotionDone AND xMotionActive THEN
            xMotionActive := FALSE;
            xMotionIssued := FALSE;

            Runtime.State := E_TrackingState.TRK_RELEASE_PRODUCT;

        // Place lỗi.
        ELSIF MotionError AND xMotionActive THEN
            xMotionActive := FALSE;

            Runtime.Response.Error := TRUE;
            Runtime.Response.ErrorID := MotionErrorID;

            Runtime.State := E_TrackingState.TRK_ERROR;
        END_IF;

    //=========================================================================
    // TRK_RELEASE_PRODUCT
    // Tắt hút, bật thổi và chuẩn bị timer.
    //=========================================================================
    E_TrackingState.TRK_RELEASE_PRODUCT:

        // Tắt hút để nhả sản phẩm.
        VacuumCommand := FALSE;

        // Bật van thổi.
        BlowCommand := TRUE;

        // Reset timer thổi trước khi vào state chờ.
        tonBlow(IN := FALSE);

        // Chuyển sang chờ đủ thời gian thổi.
        Runtime.State := E_TrackingState.TRK_WAIT_BLOW;

    //=========================================================================
    // TRK_WAIT_BLOW
    // Giữ thổi trong Config.BlowTime.
    //=========================================================================
    E_TrackingState.TRK_WAIT_BLOW:

        // Bảo đảm hút tắt.
        VacuumCommand := FALSE;

        // Giữ van thổi bật.
        BlowCommand := TRUE;

        // Chạy timer thổi.
        tonBlow(
            IN := TRUE,
            PT := Config.BlowTime
        );

        // Khi hết thời gian thổi.
        IF tonBlow.Q THEN
            // Reset timer.
            tonBlow(IN := FALSE);

            // Tắt thổi.
            BlowCommand := FALSE;

            // Đánh dấu object đã PICKED.
            Queue.Objects[Runtime.SelectedObjectIndex].State := E_TrackingObjectState.OBJ_PICKED;

            // Giải phóng cờ Reserved.
            Queue.Objects[Runtime.SelectedObjectIndex].Reserved := FALSE;

            // Giải phóng ActiveIndex.
            Queue.ActiveIndex := GVL.C_INVALID_INDEX;

            // Báo gắp thành công.
            Runtime.PickSuccess := TRUE;

            // Xóa object active trong Runtime.
            Runtime.SelectedObjectIndex := 0;
            Runtime.SelectedObjectID := 0;

            // Xóa trạng thái đã giữ vật.
            xVacuumCaptured := FALSE;

            // Phát Done.
            Runtime.Response.Done := TRUE;

            // Chuyển sang Complete.
            Runtime.State := E_TrackingState.TRK_COMPLETE;
        END_IF;

